Yaskawa INFORM job: SKRZYNIA_5340_-90_STOPNI_10BR.JBI

/JOB
//NAME SKRZYNIA_5340_-90_STOPNI_10BR
///FOLDERNAME 02-SKRZYNIE_JOBS
//POS
///NPOS 695,695,0,50,0,0
///TOOL 0
///POSTYPE PULSE
///PULSE
C00000=0,-52280,40443,0,6876,0
C00001=-82314,-24956,17040,-59626,-27382,-6248
C00002=-93910,-8625,17040,-59626,-43355,-6248
C00003=-98846,-1061,-42166,-80308,-57081,16120
C00004=-100452,6057,-48127,-85711,-56704,21322
C00005=-96957,25597,-37888,-85158,-62082,25522
C00006=-95580,33075,-33256,-84644,-64024,26851
C00007=-94380,33739,-32188,-85134,-63496,26721
C00008=-95580,33075,-33256,-84644,-64024,26851
C00009=-94940,31262,-36138,-85248,-63712,27160
C00010=-95580,33075,-33256,-84644,-64024,26851
C00011=-95263,33142,-33256,-84677,-63995,26850
C00012=-95263,33142,-33256,-84677,-63995,26850
C00013=-94261,33702,-32359,-85087,-63552,26740
C00014=-95263,33142,-33256,-84677,-63995,26850
C00015=-94777,31773,-35433,-85135,-63758,27084
C00016=-95263,33142,-33256,-84677,-63995,26850
C00017=-95260,33144,-33256,-84678,-63995,26850
C00018=-95260,33144,-33256,-84678,-63995,26850
C00019=-94282,33689,-32380,-85076,-63563,26742
C00020=-95260,33144,-33256,-84678,-63995,26850
C00021=-94827,31920,-35204,-85086,-63784,27059
C00022=-95260,33144,-33256,-84678,-63995,26850
C00023=-95258,33145,-33257,-84676,-63996,26846
C00024=-95258,33145,-33257,-84676,-63996,26846
C00025=-94286,33686,-32387,-85074,-63568,26738
C00026=-95258,33145,-33257,-84676,-63996,26846
C00027=-94874,32057,-34990,-85039,-63809,27032
C00028=-95258,33145,-33257,-84676,-63996,26846
C00029=-95258,33145,-33257,-84676,-63996,26846
C00030=-95258,33145,-33257,-84676,-63996,26846
C00031=-94323,33667,-32422,-85059,-63584,26741
C00032=-95258,33145,-33257,-84676,-63996,26846
C00033=-94899,32130,-34875,-85014,-63820,27019
C00034=-95258,33145,-33257,-84676,-63996,26846
C00035=-95258,25631,32269,-66559,-75499,2416
C00036=-95258,25631,32269,-66559,-75499,2416
C00037=-94333,26371,33350,-66433,-74983,2224
C00038=-95258,25631,32269,-66559,-75499,2416
C00039=-94886,24142,30119,-66602,-75133,2534
C00040=-95258,25631,32269,-66559,-75499,2416
C00041=-98646,19496,-17631,-99827,-80462,21224
C00042=-98811,21047,-15512,-99242,-81394,20987
C00043=-97886,21574,-14788,-99528,-80824,20997
C00044=-98811,21047,-15512,-99242,-81394,20987
C00045=-98517,19954,-17009,-99363,-81263,21101
C00046=-98811,21047,-15512,-99242,-81394,20987
C00047=-98811,19937,1242,-97498,-78933,15296
C00048=-98811,19937,1242,-97498,-78933,15296
C00049=-97933,20465,1962,-97646,-78345,15298
C00050=-98811,19937,1242,-97498,-78933,15296
C00051=-98523,18806,-285,-97586,-78782,15407
C00052=-98811,19937,1242,-97498,-78933,15296
C00053=-99152,37522,67957,-90787,-75030,-95
C00054=-99152,37522,67957,-90787,-75030,-95
C00055=-98279,38495,69612,-90504,-74443,-274
C00056=-99152,37522,67957,-90787,-75030,-95
C00057=-98708,34478,62881,-90983,-74820,488
C00058=-99152,37522,67957,-90787,-75030,-95
C00059=-98988,22776,44546,-90608,-68570,2568
C00060=-94428,854,16076,-89248,-50738,4740
C00061=-88080,-20128,-3199,-80943,-31244,2335
C00062=-50003,-39410,-5978,-16260,-18649,-25999
C00063=-48287,-44591,-17414,-16172,-14532,-25809
C00064=-85348,-13130,13838,-41209,-47455,-8220
C00065=-99199,18818,35660,-68259,-73735,6208
C00066=-95720,11094,-10147,-77005,-64537,18127
C00067=-95720,11099,-9975,-76955,-64559,18070
C00068=-97322,30100,38585,-71742,-79662,10416
C00069=-96349,30901,39804,-71630,-79090,10224
C00070=-97322,30100,38585,-71742,-79662,10416
C00071=-97054,28837,36680,-71776,-79387,10556
C00072=-97322,30100,38585,-71742,-79662,10416
C00073=-97373,30352,38967,-71736,-79717,10385
C00074=-97373,30352,38967,-71736,-79717,10385
C00075=-96432,31128,40151,-71627,-79165,10198
C00076=-97373,30352,38967,-71736,-79717,10385
C00077=-97071,28917,36802,-71776,-79407,10544
C00078=-97373,30352,38967,-71736,-79717,10385
C00079=-97356,30262,38827,-71739,-79698,10398
C00080=-97356,30262,38827,-71739,-79698,10398
C00081=-96507,30957,39891,-71642,-79201,10230
C00082=-97356,30262,38827,-71739,-79698,10398
C00083=-97092,29010,36937,-71773,-79425,10538
C00084=-97356,30262,38827,-71739,-79698,10398
C00085=-97431,30641,39402,-71725,-79780,10352
C00086=-97431,30641,39402,-71725,-79780,10352
C00087=-96578,31348,40481,-71627,-79280,10181
C00088=-97431,30641,39402,-71725,-79780,10352
C00089=-97114,29116,37095,-71767,-79448,10523
C00090=-97431,30641,39402,-71725,-79780,10352
C00091=-99739,25677,21114,-82085,-78790,-4409
C00092=-99739,25677,21114,-82085,-78790,-4409
C00093=-98872,26250,21941,-82102,-78216,-4501
C00094=-99739,25677,21114,-82085,-78790,-4409
C00095=-99422,24232,19045,-82158,-78544,-4261
C00096=-99739,25677,21114,-82085,-78790,-4409
C00097=-98070,21699,18791,-100677,-76082,-5031
C00098=-98401,27942,27737,-100067,-79473,-6121
C00099=-97586,28537,28617,-100081,-78897,-6135
C00100=-98401,27942,27737,-100067,-79473,-6121
C00101=-98064,26400,25481,-100144,-79339,-5917
C00102=-98401,27942,27737,-100067,-79473,-6121
C00103=-99160,29228,35009,-99418,-79080,-8034
C00104=-98369,30564,38686,-99156,-78226,-8682
C00105=-97572,31199,39655,-99108,-77655,-8715
C00106=-98369,30564,38686,-99156,-78226,-8682
C00107=-98044,28949,36247,-99232,-78106,-8445
C00108=-98369,30564,38686,-99156,-78226,-8682
C00109=-99160,29228,35009,-99418,-79080,-8034
C00110=-98369,30564,38686,-99156,-78226,-8682
C00111=-97572,31199,39655,-99108,-77655,-8715
C00112=-98369,30564,38686,-99156,-78226,-8682
C00113=-98044,28949,36247,-99232,-78106,-8445
C00114=-98369,30564,38686,-99156,-78226,-8682
C00115=-91461,-11352,-34112,-115843,-54659,7933
C00116=-98486,-14751,-40891,-114294,-59712,7739
C00117=-84089,-24462,-58822,-138905,-52068,17717
C00118=-93370,-29108,-64994,-133695,-56362,15444
C00119=-62749,-65297,-81682,-146767,-31843,20298
C00120=-73187,-23116,26488,-26118,-57509,-28469
C00121=-99665,-12992,-24886,-73613,-54905,-950
C00122=-98398,-8109,-25057,-81551,-55130,4513
C00123=-99451,17861,2757,-80571,-73406,6045
C00124=-99819,33446,48735,-87787,-79679,-1235
C00125=-99819,33446,48735,-87787,-79679,-1235
C00126=-98945,34179,49898,-87659,-79086,-1350
C00127=-99819,33446,48735,-87787,-79679,-1235
C00128=-99591,32133,46677,-87830,-79529,-1033
C00129=-99819,33446,48735,-87787,-79679,-1235
C00130=-98853,28116,28355,-96898,-79749,4777
C00131=-98853,30464,37910,-96149,-78952,2546
C00132=-98284,30904,38579,-96116,-78548,2515
C00133=-98853,30464,37910,-96149,-78952,2546
C00134=-98656,29478,36421,-96191,-78865,2688
C00135=-98853,30464,37910,-96149,-78952,2546
C00136=-94437,3365,15121,-90804,-55123,21
C00137=-76606,-19838,2636,-59027,-23020,-13375
C00138=-49667,-45532,-21960,-5654,-17518,-35856
C00139=-47485,-50287,-32535,-1070,-13732,-37871
C00140=-36103,-65917,11738,-26975,4295,7905
C00141=6327,-52297,40484,-8600,6957,5944
C00142=0,-52280,40443,0,6876,0
C00143=0,-52280,40443,0,6876,0
C00144=0,-43112,23163,32261,-40956,29092
C00145=-48283,-21883,28214,-25170,-26491,48363
C00146=-46664,-3144,58041,-18842,-32105,45325
C00147=-50347,-18571,12268,-49104,-16423,60029
C00148=-53571,-17125,12073,-56866,-17385,63433
C00149=-52069,-15730,13206,-55612,-16432,62999
C00150=-53474,-15384,13495,-57637,-17161,63825
C00151=-53571,-17125,12073,-56866,-17385,63433
C00152=-50509,-19000,10610,-51503,-15997,61182
C00153=-53130,-17211,12007,-56251,-17152,63186
C00154=-51822,-15992,12994,-55136,-16324,62798
C00155=-53635,-15431,13457,-57815,-17251,63894
C00156=-53130,-17211,12007,-56251,-17152,63186
C00157=-50704,-18403,11069,-52157,-16018,61478
C00158=-53231,-16470,14622,-53206,-17893,61673
C00159=-51756,-15101,15744,-51790,-16990,61165
C00160=-53741,-14453,16285,-54808,-17949,62397
C00161=-53231,-17580,11714,-56182,-17246,63139
C00162=-51814,-19410,10295,-53186,-16720,61844
C00163=-53629,-18979,7405,-62018,-16535,65958
C00164=-52238,-17698,8415,-61175,-15613,65699
C00165=-53551,-17401,8655,-62910,-16346,66402
C00166=-52880,-17654,11656,-55678,-17066,62935
C00167=-51005,-17995,11387,-52847,-16122,61778
C00168=-52964,-17611,11689,-55811,-17106,62990
C00169=-51611,-16353,12697,-54642,-16249,62582
C00170=-53495,-15765,13180,-57466,-17201,63739
C00171=-52964,-17611,11689,-55811,-17106,62990
C00172=-51030,-17982,11395,-52891,-16135,61798
C00173=-52975,-17563,11726,-55850,-17109,63009
C00174=-51607,-16289,12749,-54669,-16241,62596
C00175=-53283,-15811,13140,-57177,-17094,63622
C00176=-52975,-17563,11726,-55850,-17109,63009
C00177=-50945,-18019,11363,-52741,-16103,61737
C00178=-52728,-17788,11545,-55393,-17010,62816
C00179=-51045,-16207,12813,-53894,-15944,62287
C00180=-52895,-15647,13274,-56746,-16874,63461
C00181=-52728,-17788,11545,-55393,-17010,62816
C00182=-50945,-18019,11363,-52741,-16103,61737
C00183=-52556,-17520,11756,-55311,-16888,62798
C00184=-51113,-16157,12849,-54025,-15975,62343
C00185=-52730,-15718,13210,-56498,-16792,63358
C00186=-52556,-17520,11756,-55311,-16888,62798
C00187=-50945,-18019,11363,-52741,-16103,61737
C00188=-51893,-17787,11546,-54246,-16568,62356
C00189=-50379,-16341,12703,-52826,-15610,61849
C00190=-52406,-15704,13225,-56071,-16614,63190
C00191=-51893,-17787,11546,-54246,-16568,62356
C00192=-50028,-22953,-3957,-22347,-31919,54220
C00193=-50947,-22502,-3625,-23433,-32061,54736
C00194=-49421,-20951,-2455,-21951,-31329,54057
C00195=-51207,-20433,-2055,-24026,-31698,55041
C00196=-50529,-22709,-3778,-22940,-31995,54502
C00197=-49763,-25421,-36239,-24565,-26935,60445
C00198=-49763,-25421,-36239,-24565,-26935,60445
C00199=-48299,-23485,-34758,-23276,-26122,59713
C00200=-50218,-22723,-34165,-25568,-26529,60993
C00201=-49763,-25421,-36239,-24565,-26935,60445
C00202=-50713,-12366,-58367,-41124,-17813,74400
C00203=-50824,-12254,-58263,-41255,-17847,74484
C00204=-49431,-10052,-56192,-40383,-17131,73813
C00205=-50915,-9358,-55524,-41955,-17664,74847
C00206=-51028,-12852,-58814,-41301,-17980,74542
C00207=-49763,-25421,-36239,-24565,-26935,60445
C00208=-50529,-22709,-3778,-22940,-31995,54502
C00209=-45389,-28224,4312,-35967,-15579,54278
C00210=-40154,-51179,-915,-24203,-8234,36524
C00211=0,-52280,40443,0,6876,0
C00212=0,-52280,40443,0,6876,0
C00213=-2117,-50103,-33543,-4117,45077,85249
C00214=26439,-48928,-33543,-4117,-52362,85249
C00215=26439,-27355,-33543,-41485,-52362,85249
C00216=39218,-24492,-41653,-51934,-39374,86964
C00217=39218,-24492,-41653,-51934,-39374,86964
C00218=46639,7575,-9331,-26045,-41627,82486
C00219=47278,8641,-9483,-26175,-40625,82510
C00220=46369,10567,-7126,-26545,-41054,82831
C00221=47278,8641,-9483,-26175,-40625,82510
C00222=48256,9506,-8430,-25641,-40400,82076
C00223=47278,8641,-9483,-26175,-40625,82510
C00224=44522,-635,-31983,-49264,-28311,89687
C00225=44247,-628,-31975,-49394,-28443,89790
C00226=43310,1314,-29842,-49807,-28910,90140
C00227=44247,-628,-31975,-49394,-28443,89790
C00228=45313,152,-31124,-48894,-27920,89380
C00229=44247,-628,-31975,-49394,-28443,89790
C00230=41572,-13073,-22520,-50760,-38355,84033
C00231=21909,-6773,-14577,-94161,-56302,89381
C00232=23773,-3183,-10897,-94486,-55065,89563
C00233=24904,-823,-8382,-94654,-54308,89644
C00234=24395,1151,-6219,-94590,-54651,89617
C00235=24904,-823,-8382,-94654,-54308,89644
C00236=26178,-337,-7854,-94816,-53451,89710
C00237=24904,-823,-8382,-94654,-54308,89644
C00238=17020,-16061,-23281,-93084,-59494,88637
C00239=-21568,-26506,-31664,-90508,-85573,86639
C00240=-8557,-39769,-22319,-51419,-69406,84680
C00241=-8557,-39769,-22319,-51419,-69406,84680
C00242=32994,-9735,-10751,-29019,-59471,69498
C00243=43974,9628,-22604,-36190,-36396,73426
C00244=45932,13115,-22315,-37472,-33732,73846
C00245=45228,14664,-20329,-37571,-34159,74020
C00246=45932,13115,-22315,-37472,-33732,73846
C00247=46653,13731,-21526,-37109,-33514,73520
C00248=45932,13115,-22315,-37472,-33732,73846
C00249=39039,866,-6986,-42761,-44691,67687
C00250=30717,-9248,-22721,-77433,-42696,79486
C00251=32434,-7077,-20587,-77571,-41526,79457
C00252=31883,-5576,-19073,-77676,-41878,79560
C00253=32434,-7077,-20587,-77571,-41526,79457
C00254=33092,-6769,-20280,-77576,-41084,79417
C00255=32434,-7077,-20587,-77571,-41526,79457
C00256=30527,-14106,-27266,-76898,-42917,79150
C00257=25454,-9581,-17335,-94425,-53880,89429
C00258=24965,-2445,-10120,-94645,-54263,89631
C00259=24893,-1278,-8874,-94650,-54314,89639
C00260=24417,557,-6877,-94595,-54636,89618
C00261=24893,-1278,-8874,-94650,-54314,89639
C00262=25752,-956,-8526,-94759,-53737,89684
C00263=24893,-1278,-8874,-94650,-54314,89639
C00264=23817,-1527,-9142,-94518,-55040,89587
C00265=24871,-1152,-8735,-94651,-54328,89643
C00266=24440,508,-6926,-94601,-54619,89624
C00267=24871,-1152,-8735,-94651,-54328,89643
C00268=25635,-865,-8427,-94748,-53815,89684
C00269=24871,-1152,-8735,-94651,-54328,89643
C00270=33203,-4295,-13750,-123758,-49995,81034
C00271=35028,4195,-6818,-132965,-58836,87950
C00272=35028,4195,-6818,-132965,-58836,87950
C00273=34452,5837,-4911,-132720,-59045,87770
C00274=35028,4195,-6818,-132965,-58836,87950
C00275=35710,4593,-6360,-133217,-58512,88125
C00276=35028,4195,-6818,-132965,-58836,87950
C00277=24762,-11408,-28656,-113055,-60293,85383
C00278=-28645,-26349,-41223,-103369,-91870,78302
C00279=-28645,-26349,-41223,-103369,-91870,78302
C00280=-25549,-24286,-26215,-66769,-87032,80148
C00281=27561,-8271,-12315,-63268,-52553,74387
C00282=29336,-165,-3925,-63163,-51316,74265
C00283=29518,765,-2904,-63127,-51205,74233
C00284=28850,2962,-447,-63227,-51636,74327
C00285=29518,765,-2904,-63127,-51205,74233
C00286=30662,1292,-2320,-62902,-50501,74035
C00287=29518,765,-2904,-63127,-51205,74233
C00288=30773,10953,32136,-106912,-46141,83783
C00289=30773,10953,32136,-106912,-46141,83783
C00290=30080,13410,35293,-106601,-46463,83481
C00291=30773,10953,32136,-106912,-46141,83783
C00292=32007,11622,32987,-106899,-45346,83915
C00293=30773,10953,32136,-106912,-46141,83783
C00294=28321,-8642,-16372,-95739,-47180,89965
C00295=28583,-7344,-15096,-95864,-47019,90043
C00296=27897,-5229,-12965,-95873,-47499,90079
C00297=28583,-7344,-15096,-95864,-47019,90043
C00298=29900,-6813,-14567,-96101,-46141,90154
C00299=28583,-7344,-15096,-95864,-47019,90043
C00300=27852,-7537,-15286,-95742,-47508,89986
C00301=28448,-7306,-15058,-95845,-47110,90035
C00302=27795,-5283,-13021,-95851,-47567,90065
C00303=28448,-7306,-15058,-95845,-47110,90035
C00304=29772,-6774,-14527,-96083,-46226,90146
C00305=28448,-7306,-15058,-95845,-47110,90035
C00306=18552,-19531,-26179,-93438,-53589,88597
C00307=40301,-14999,-52277,-148979,-69262,86714
C00308=42323,-33,-37432,-150113,-69667,87489
C00309=53245,19091,3515,-165691,-72595,90030
C00310=53641,19552,4138,-165817,-72473,90151
C00311=53058,20743,5761,-165615,-72317,89948
C00312=53641,19552,4138,-165817,-72473,90151
C00313=54155,20160,4967,-165982,-72308,90306
C00314=53641,19552,4138,-165817,-72473,90151
C00315=23439,-10154,-17205,-109204,-58547,76547
C00316=2382,-21913,-40813,-107544,-74451,77239
C00317=-31257,-15877,-35733,-102288,-96107,74463
C00318=-39204,-18003,-7668,-86141,-99190,68413
C00319=-5592,-5690,18047,-75373,-79525,63129
C00320=19039,-439,25862,-68224,-64120,61443
C00321=21624,5223,26011,-69375,-61155,63193
C00322=24437,11840,34139,-68260,-59598,62567
C00323=24053,13588,36402,-68249,-59917,62491
C00324=24437,11840,34139,-68260,-59598,62567
C00325=25079,12112,34488,-68051,-59212,62472
C00326=24437,11840,34139,-68260,-59598,62567
C00327=21370,4935,25667,-69451,-61310,63230
C00328=-18351,-11002,3811,-80352,-86206,66275
C00329=-34619,-5846,8788,-82342,-97004,67025
C00330=-40684,-19963,-8478,-86482,-100204,67987
C00331=1570,-13136,-5998,-86227,-71173,69099
C00332=13966,-6596,-2340,-86587,-62612,70052
C00333=24093,-1862,-9504,-94546,-54850,89594
C00334=24093,-1862,-9504,-94546,-54850,89594
C00335=23519,425,-7024,-94488,-55240,89573
C00336=24093,-1862,-9504,-94546,-54850,89594
C00337=25256,-1442,-9053,-94693,-54067,89656
C00338=24093,-1862,-9504,-94546,-54850,89594
C00339=27718,4364,12871,-105518,-51077,86669
C00340=27718,4364,12871,-105518,-51077,86669
C00341=27164,6353,15202,-105385,-51398,86539
C00342=27718,4364,12871,-105518,-51077,86669
C00343=28828,4851,13441,-105618,-50355,86801
C00344=27718,4364,12871,-105518,-51077,86669
C00345=20930,-1364,27707,-95004,-52134,77785
C00346=-41463,-32191,18163,-91991,-64949,55938
C00347=0,-52277,40442,0,6872,4
C00348=-82314,-24956,17040,-59626,-27382,-6248
C00349=-93910,-8625,17040,-59626,-43355,-6248
C00350=-98846,-1061,-42166,-80308,-57081,16120
C00351=-100452,6057,-48127,-85711,-56704,21322
C00352=-95564,34698,-34234,-85516,-63941,27819
C00353=-94221,34299,-28769,-82558,-65564,25844
C00354=-94107,37241,-30442,-84005,-65307,27544
C00355=-95103,32620,-31323,-83378,-64939,26072
C00356=-95103,32620,-31323,-83378,-64939,26072
C00357=-93990,32828,-31380,-83932,-64473,26160
C00358=-94063,31710,-30585,-83283,-64598,25457
C00359=-96692,32939,-31211,-82617,-65723,26190
C00360=-96111,21840,170,-71736,-70232,11396
C00361=-94229,22391,773,-71789,-70557,11468
C00362=-94283,22521,1025,-71678,-70686,11433
C00363=-95675,19167,-4176,-72970,-68231,11735
C00364=-95681,24338,3488,-71459,-71669,11415
C00365=-94245,22750,1246,-71757,-70674,11453
C00366=-94341,22923,1499,-71729,-70746,11440
C00367=-96213,24222,3324,-71394,-71999,11479
C00368=-95517,23330,2066,-71543,-71508,11507
C00369=-94304,22892,1449,-71738,-70721,11443
C00370=-94158,22889,1452,-71756,-70627,11429
C00371=-96071,24319,3461,-71408,-71916,11455
C00372=-96941,-6406,-33809,-76117,-54125,10511
C00373=-89093,-33107,-44597,-67545,-52550,2722
C00374=-66103,-61757,7450,-21008,-32955,-5749
C00375=4223,-52290,40457,-5766,6913,3980
C00376=4223,-52290,40457,-5766,6913,3980
C00377=-4538,-50065,-33535,-3011,44998,84219
C00378=24207,-49248,-33668,-5551,-52644,86091
C00379=25094,-27722,-33812,-41887,-53054,85599
C00380=38036,-25052,-42086,-52219,-40087,87228
C00381=37328,-2824,-24733,-57182,-37821,90318
C00382=36700,-2520,-13735,-51589,-42201,86442
C00383=37520,2330,-3498,-48550,-43875,84431
C00384=37520,1020,-12079,-52650,-40851,87066
C00385=48458,-261,-12985,-24069,-43340,80504
C00386=36153,7296,-1758,-40139,-50302,89334
C00387=37146,11264,2520,-40849,-50296,89553
C00388=38059,11410,-1863,-40565,-47910,90206
C00389=36726,6476,-7858,-41213,-48206,90783
C00390=19339,7883,9818,-77509,-64249,74140
C00391=19027,1888,-16187,-103553,-67480,82955
C00392=24158,3537,-14322,-106039,-60939,84018
C00393=24143,4321,-7309,-103852,-59670,81875
C00394=19531,2904,-8928,-102027,-65985,80961
C00395=20232,-3383,-14682,-86495,-63009,78978
C00396=-24375,-51634,-49601,-83793,-94064,73950
C00397=4223,-52290,40457,-5766,6913,3980
C00398=-4825,-36686,24602,37792,-30278,35378
C00399=-46221,-29633,7403,-27051,-24124,46751
C00400=-46221,-29633,7403,-27051,-24124,46751
C00401=-52474,-20611,11454,-41004,-23045,52959
C00402=-60257,-19980,-2088,-84190,-23320,82051
C00403=-63868,-19883,-6318,-95759,-28031,88346
C00404=-51819,-22965,8574,-41365,-22900,53139
C00405=-4825,-36686,24602,37792,-30278,35378
C00406=0,-52280,40443,0,6876,0
C00407=4223,-52290,40457,-5766,6913,3980
C00408=-66103,-61757,7450,-21008,-32955,-5749
C00409=-89093,-33107,-44597,-67545,-52550,2722
C00410=-96941,-6406,-33809,-76117,-54125,10511
C00411=-99429,14378,84,-80785,-71596,8628
C00412=-99699,24313,24829,-82602,-77917,4569
C00413=-98066,26841,20697,-83331,-79245,6860
C00414=-98079,26929,20513,-83349,-79351,6953
C00415=-99638,19663,10292,-84193,-74452,7551
C00416=-99636,19665,10291,-84197,-74448,7550
C00417=-98131,26698,20177,-83371,-79212,6975
C00418=-98097,25980,12653,-84102,-79057,9159
C00419=-99636,19665,10291,-84197,-74448,7550
C00420=-99636,19665,10291,-84197,-74448,7550
C00421=-98186,26934,20517,-83350,-79332,6954
C00422=-98240,27087,20738,-83333,-79465,6940
C00423=-99636,19665,10291,-84197,-74448,7550
C00424=-99215,3992,8526,-80547,-63068,1835
C00425=-100264,1107,23397,-72827,-59854,-5092
C00426=-100264,1107,23397,-72827,-59854,-5092
C00427=-99514,-9483,18258,-71284,-60958,-4118
C00428=-61441,-38616,11032,-55510,-42874,-3049
C00429=4223,-52290,40457,-5766,6913,3980
C00430=-22331,-23394,-30093,-82917,-82006,85712
C00431=22434,-14401,-3235,-51104,-60845,74728
C00432=42744,21307,45077,-24753,-69813,65333
C00433=33655,14083,18147,-45417,-58301,71861
C00434=33641,11943,8279,-47835,-54840,73983
C00435=36574,13250,23432,-35354,-61822,69159
C00436=28497,326,20939,-70981,-47632,72427
C00437=30972,5983,29862,-68494,-46670,70994
C00438=31029,11571,45127,-63398,-49004,67378
C00439=28971,8096,39948,-65070,-49810,68216
C00440=29759,-12862,-24221,-91747,-41905,86600
C00441=35278,-10419,-21940,-93284,-36771,87139
C00442=36208,-10883,-22374,-93618,-35345,87231
C00443=27219,-23595,-33313,-89555,-43517,85303
C00444=10564,-40773,-45889,-85382,-54876,82708
C00445=-14984,-61618,-24572,-87392,-53367,60735
C00446=9346,-67436,-18786,-75708,-34590,53709
C00447=40938,-55232,35946,-9746,5421,6718
C00448=4223,-52290,40457,-5766,6913,3980
C00449=-4825,-36686,24602,37792,-30278,35378
C00450=-46221,-29633,7403,-27051,-24124,46751
C00451=-56796,-22932,368,-68953,-21567,70907
C00452=-61611,-20349,-6598,-95791,-25091,88405
C00453=-63740,-19715,-7390,-98604,-28245,90373
C00454=-52085,-22687,8760,-40927,-22666,52970
C00455=-49294,-34086,9663,-30689,-30758,52546
C00456=4223,-52290,40457,-5766,6913,3980
C00457=0,-52280,40443,0,6876,0
C00458=0,-52280,40443,0,6876,0
C00459=-61754,-61602,7279,-16215,-32140,-7126
C00460=-89313,-24027,20291,-53466,-58905,-4975
C00461=-97807,-25409,-21837,-78881,-62828,2121
C00462=-95644,-21015,-18476,-76474,-46020,1039
C00463=-99784,20282,11129,-84157,-74554,7499
C00464=-100058,25789,39872,-88643,-74345,1113
C00465=-98402,30585,40634,-89771,-78826,2411
C00466=-98157,28480,31016,-94616,-79375,5454
C00467=-99711,20530,18234,-96341,-74733,7105
C00468=-100058,25789,39872,-88643,-74345,1113
C00469=-98402,30585,40634,-89771,-78826,2411
C00470=-98157,28480,31016,-94616,-79375,5454
C00471=-99711,20530,18234,-96341,-74733,7105
C00472=-99082,-18510,-57081,-109378,-57172,19856
C00473=-62624,-58412,-72925,-116868,-19429,18539
C00474=-75165,-16680,32803,-38944,-52307,-27215
C00475=-75165,-16680,32803,-38944,-52307,-27215
C00476=-96391,11374,61850,-52875,-60261,-22353
C00477=-96391,-17993,-25254,-79577,-45337,-1997
C00478=-84714,-13514,-21320,-79690,-37366,-2300
C00479=-92093,-5454,-13554,-80916,-52292,-613
C00480=-99761,24721,23429,-79408,-77929,-316
C00481=-100093,22783,4772,-83722,-77198,5432
C00482=-98451,25119,10323,-84368,-78687,2343
C00483=-98528,26732,19657,-84000,-79459,-654
C00484=-100109,23919,19160,-82044,-77303,1139
C00485=-98037,-4340,-16930,-86109,-58746,2389
C00486=-93345,-31758,-40240,-83703,-37467,-946
C00487=-81087,-35886,-14825,-53529,-36311,-18004
C00488=-47029,-49867,-20464,-11808,-29290,-36568
///LIMIT ON
C00489=-41431,-67449,10869,-1325,127,-6150
///LIMIT OFF
C00490=6328,-52297,40483,-8599,6957,5944
C00491=-8648,-69005,-18270,-84275,-43232,53472
C00492=18757,-59462,-34892,-84638,-37529,67311
C00493=26772,-23733,-33422,-89486,-43820,85275
C00494=29039,-10071,-21608,-91386,-45181,86629
C00495=29639,-5923,-17523,-91591,-45648,86808
C00496=29709,-5453,-17046,-91618,-45636,86826
C00497=29138,-10182,-21714,-91372,-45196,86624
C00498=20424,-22725,-32635,-88800,-51006,85261
C00499=28416,-11420,-25238,-98178,-46636,84572
C00500=30481,-6584,-16425,-92636,-44382,82541
C00501=30464,-7521,-23523,-96665,-44944,85234
C00502=28416,-11420,-25238,-98178,-46636,84572
C00503=-23524,-33387,-42654,-89891,-81168,80229
C00504=-23524,-33387,-42654,-89891,-81168,80229
C00505=33935,-6399,-10013,-60506,-43064,77980
C00506=34878,-3211,-6740,-60356,-42422,77865
C00507=34873,-3218,-6748,-60357,-42424,77868
C00508=33935,-6399,-10013,-60506,-43064,77980
C00509=17782,-19597,1250,-60925,-51448,69151
C00510=-243,-43047,-13224,-69794,-55957,65877
C00511=42700,-55269,36176,-13619,5333,9062
C00512=6328,-52297,40483,-8599,6957,5944
C00513=-10231,-60460,6271,71658,-11927,-13637
C00514=-49129,-39322,3023,-34904,-18609,43900
C00515=-57258,-19535,13114,-46502,-25798,55150
C00516=-58736,-19151,1344,-78268,-22199,76919
C00517=-56868,-17231,8572,-62431,-21728,66645
C00518=-56011,-29317,6725,-41009,-27363,52457
C00519=-10137,-60963,4526,62308,-14518,-6745
C00520=0,-52280,40443,0,6876,0
C00521=0,-52280,40443,0,6876,0
C00522=-41653,-63035,2931,-3578,-7576,-14589
C00523=-45770,-50109,-20524,-10089,-29273,-37310
C00524=-80544,-36303,-15042,-52975,-36116,-18265
C00525=-93028,-32302,-40599,-83495,-37263,-1079
C00526=-98446,-3141,-15678,-86094,-59021,2414
C00527=-99951,24070,19376,-82000,-77829,1145
C00528=-98655,27908,24922,-81730,-79774,792
C00529=-98593,28720,26118,-81685,-80145,709
C00530=-99951,24070,19376,-82000,-77829,1145
C00531=-99951,24070,19376,-82000,-77829,1145
C00532=-98577,27118,23759,-81796,-79157,859
C00533=-98518,28577,26461,-81649,-79882,537
C00534=-99951,24070,19376,-82000,-77829,1145
C00535=-99951,24070,19376,-82000,-77829,1145
C00536=-98479,26563,22955,-81844,-78651,906
C00537=-98651,28095,26058,-81646,-79654,489
C00538=-99951,24070,19376,-82000,-77829,1145
C00539=-97595,-1409,-12320,-84284,-60474,1798
C00540=-100010,-16422,-27011,-84227,-53565,945
C00541=-88098,-29848,-22776,-71580,-48483,-7812
C00542=-81694,-37220,-20464,-64791,-45723,-12569
C00543=-45770,-50109,-20524,-10089,-29273,-37310
C00544=-40984,-65135,6743,-2520,-4051,-10897
C00545=0,-52280,40443,0,6876,0
C00546=40939,-55232,35946,-9746,5421,6719
C00547=8707,-69002,-18268,-75213,-34271,52581
C00548=23267,-58917,-25142,-81990,-31707,62852
C00549=27307,-5613,10331,-81857,-46454,76095
C00550=30064,-5598,-963,-91827,-44222,81590
C00551=30419,-1725,5291,-88668,-43977,80354
C00552=30554,-300,10432,-88528,-43656,79164
C00553=29815,-6351,-3652,-90193,-44535,81892
C00554=29567,1847,27834,-65726,-48411,69959
C00555=23257,11670,30420,-81328,-57342,77033
C00556=23257,16856,45442,-77525,-58254,73578
C00557=21577,7912,33836,-78698,-59121,74340
C00558=17856,-9033,24892,-70658,-55966,67475
C00559=20838,-7097,2019,-111788,-62648,79114
C00560=40635,280,-7982,-142398,-56681,90238
C00561=32653,-9455,434,-90251,-40347,77213
C00562=40635,572,-6271,-142064,-55879,89947
C00563=40665,7761,2001,-141975,-55632,89869
C00564=40707,9678,10648,-140211,-51894,88431
C00565=39416,1907,3178,-139370,-51839,87774
C00566=7767,-21333,-19174,-120411,-69473,77116
C00567=33666,-18553,20064,-54519,-41956,59729
C00568=4032,-43511,13506,-33366,-30942,40837
C00569=22997,-56875,21315,16958,-8102,3163
C00570=0,-52280,40443,0,6876,0
C00571=-50974,-46557,23391,-77768,-13896,42026
C00572=-53474,-39983,4253,-39182,-18848,44272
C00573=-56619,-19856,12878,-45665,-25558,54806
C00574=-53298,-26712,-11188,-26889,-32979,52528
C00575=-57200,-20845,-7559,-37425,-33513,53351
C00576=-58648,-23818,-25853,-45100,-31207,62168
C00577=-58477,-22145,-38977,-48305,-29254,64725
C00578=-51868,-27423,-11673,-25269,-32728,51737
C00579=-49121,-45409,-2608,-26656,-19965,38583
C00580=-21301,-61008,4568,43957,-10534,-712
C00581=0,-52280,40443,0,6876,0
C00582=0,-52280,40443,0,6876,0
C00583=-40221,-67507,11044,-1325,-65,-6716
C00584=-45770,-50109,-20525,-10088,-29274,-37311
C00585=-80544,-36303,-15042,-52975,-36116,-18265
C00586=-93028,-32301,-40599,-83495,-37262,-1079
C00587=-97841,-4898,-17503,-86112,-58614,2374
C00588=-98519,17635,7561,-106659,-77043,7343
C00589=-96245,23653,15791,-106069,-78604,6508
C00590=-96042,26225,19489,-105739,-79656,6032
C00591=-98519,17635,7561,-106659,-77043,7343
C00592=-98519,17635,7561,-106659,-77043,7343
C00593=-96298,25666,18652,-105800,-79560,6117
C00594=-95268,26547,15396,-109206,-81354,7908
C00595=-98519,17635,7561,-106659,-77043,7343
C00596=-96138,5697,-7380,-109479,-68538,9618
C00597=-100287,-3253,-24038,-111364,-68562,12025
C00598=-99412,-19117,-26908,-100833,-57247,5735
C00599=-91712,-30589,-22890,-72058,-50969,-7685
C00600=-81694,-37221,-20464,-64791,-45723,-12569
C00601=-45770,-50109,-20525,-10088,-29274,-37311
C00602=-40221,-67507,11044,-1325,-65,-6716
C00603=0,-52280,40443,0,6876,0
C00604=51241,-30653,28678,4016,-29070,6398
C00605=46185,-61941,-37286,-12736,-10732,51851
C00606=-13205,-44768,-23966,-65315,-59418,73750
C00607=-11120,-40541,-20876,-69249,-61539,75403
C00608=-836,-13033,12361,-83908,-73576,73378
C00609=18912,6214,32354,-79489,-60743,73080
C00610=21217,10898,38129,-78632,-59343,72736
C00611=23447,16313,45262,-77527,-58074,72177
C00612=23610,23756,64158,-73325,-59549,68283
C00613=18912,6214,32354,-79489,-60743,73080
C00614=-836,-13033,12361,-83908,-73576,73378
C00615=-20209,-39682,-20467,-71924,-67122,76479
C00616=-20209,-39682,-20467,-71924,-67122,76479
C00617=26353,-3691,11741,-61723,-54035,71160
C00618=29598,-2090,11073,-69087,-47235,76987
C00619=30217,-1844,4641,-75777,-45517,79979
C00620=29529,1742,11379,-68166,-49318,73572
C00621=24010,-9039,-4437,-79986,-50972,77255
C00622=24652,-10740,-12845,-99298,-50700,81949
C00623=28976,-2672,-4778,-100308,-47937,82653
C00624=31030,-2921,-9996,-112394,-49006,86348
C00625=24652,-10740,-12845,-99298,-50700,81949
C00626=-25637,-26222,-38592,-96633,-85474,81576
C00627=-36771,-16470,-4689,-95304,-89579,74076
C00628=-33704,-12343,7746,-85568,-87064,70052
C00629=4032,-43511,13506,-33366,-30942,40837
C00630=27500,-60047,23168,28912,-2679,-5784
C00631=0,-52280,40443,0,6876,0
C00632=-50971,-46557,23390,-77766,-13895,42026
C00633=-53475,-39984,4253,-39182,-18848,44273
C00634=-56619,-19856,12878,-45665,-25558,54806
C00635=-57643,-27958,-8553,-51854,-24771,59787
C00636=-66195,-24410,-19095,-90567,-31132,85904
C00637=-63290,-24193,-14362,-80030,-27547,78073
C00638=-39040,-40975,-15408,-18643,-21575,44866
C00639=-11647,-69843,-10959,56399,-11165,-4616
C00640=-15394,-57237,30542,-10392,5525,8219
C00641=0,-52280,40443,0,6876,0
C00642=0,-52280,40443,0,6876,0
///LIMIT ON
C00643=-40221,-67507,11044,-1325,-65,-6716
///LIMIT OFF
C00644=-45770,-50109,-20525,-10088,-29274,-37311
C00645=-95022,-19559,-3970,-66108,-42168,-11789
C00646=-84972,-7110,7117,-67721,-41324,-10731
C00647=-83869,-8155,6098,-67213,-40658,-10968
C00648=-99927,21772,-3530,-88309,-78218,7709
C00649=-97220,21950,1672,-79686,-74035,6807
C00650=-96918,21734,-3846,-80685,-73375,8528
C00651=-99839,23064,19027,-85806,-76881,822
C00652=-99839,23064,19027,-85806,-76881,822
C00653=-98572,26113,23382,-85571,-78492,509
C00654=-98656,28006,28806,-88976,-79248,97
C00655=-99839,24479,25828,-85077,-77001,-891
C00656=-99133,24879,24637,-94741,-77121,-2989
C00657=-98191,27052,27787,-94567,-78528,-3332
C00658=-98227,29022,36334,-93788,-77894,-5388
C00659=-100426,22466,21877,-95586,-77332,-2808
C00660=-99839,23064,19027,-85806,-76881,822
C00661=-86774,-13232,-16630,-85484,-41019,-1154
C00662=-97999,-21060,-29835,-88214,-48653,956
C00663=-98846,-3268,25064,-74217,-51189,-12584
C00664=-70313,-35289,-4922,-51188,-38634,-20596
C00665=-81694,-37221,-20464,-64791,-45723,-12569
C00666=-45770,-50109,-20525,-10088,-29274,-37311
C00667=-41628,-63095,3038,-3547,-7472,-14475
C00668=4223,-52290,40457,-5766,6913,3980
C00669=4224,-52288,40457,-5773,6909,3978
C00670=4224,-52288,40457,-28770,-64753,45638
C00671=6548,2882,44080,-77825,-67624,70557
C00672=22702,21750,69443,-66118,-61597,67582
C00673=25585,21999,63350,-62249,-61285,68688
C00674=25777,17209,50811,-62979,-59886,70957
C00675=23226,22825,71113,-65575,-61542,67353
C00676=24931,14697,51677,-80718,-51653,72069
C00677=24746,14409,39758,-87518,-53542,76879
C00678=24784,21556,58944,-82031,-53873,72431
C00679=22657,12722,42993,-85587,-54940,74916
C00680=-4427,-20395,-7318,-104668,-69521,79317
C00681=768,-20151,-3587,-97758,-65802,76626
C00682=-14736,-21545,-1233,-93598,-60476,72578
C00683=1642,-46684,14475,-47609,-24983,34912
C00684=27500,-60047,23168,28912,-2679,-5784
C00685=0,-52280,40443,0,6876,0
C00686=-50971,-46557,23390,-77766,-13895,42026
C00687=-53475,-39984,4253,-39182,-18848,44273
C00688=-56619,-19856,12878,-45665,-25558,54806
C00689=-53891,-17708,14512,-43170,-23995,53902
C00690=-60674,-17500,6427,-71116,-24772,71097
C00691=-63181,-17997,2063,-82122,-26831,78394
C00692=-39402,-27697,7664,-17904,-21663,43170
C00693=-11647,-69843,-10959,56399,-11165,-4616
C00694=0,-52280,40443,0,6876,0
BC00000=464364
BC00001=445130
BC00002=445130
BC00003=445130
BC00004=445130
BC00005=445130
BC00006=445130
BC00007=445130
BC00008=445130
BC00009=445130
BC00010=445130
BC00011=491232
BC00012=491232
BC00013=491232
BC00014=491232
BC00015=491232
BC00016=491232
BC00017=537442
BC00018=537442
BC00019=537442
BC00020=537442
BC00021=537442
BC00022=537442
BC00023=583546
BC00024=583546
BC00025=583546
BC00026=583546
BC00027=583546
BC00028=583546
BC00029=606594
BC00030=606594
BC00031=606594
BC00032=606594
BC00033=606594
BC00034=606594
BC00035=559393
BC00036=559393
BC00037=559393
BC00038=559393
BC00039=559393
BC00040=559393
BC00041=605503
BC00042=605503
BC00043=605504
BC00044=605503
BC00045=605503
BC00046=605503
BC00047=605503
BC00048=605503
BC00049=605503
BC00050=605503
BC00051=605503
BC00052=605503
BC00053=604255
BC00054=604255
BC00055=604255
BC00056=604255
BC00057=604255
BC00058=604255
BC00059=604255
BC00060=604255
BC00061=604255
BC00062=604255
BC00063=699121
BC00064=714117
BC00065=714117
BC00066=743139
BC00067=742930
BC00068=721797
BC00069=721797
BC00070=721797
BC00071=721797
BC00072=721797
BC00073=737203
BC00074=737203
BC00075=737203
BC00076=737203
BC00077=737203
BC00078=737203
BC00079=783275
BC00080=783275
BC00081=783275
BC00082=783275
BC00083=783275
BC00084=783275
BC00085=806364
BC00086=806364
BC00087=806364
BC00088=806364
BC00089=806364
BC00090=806364
BC00091=843190
BC00092=843190
BC00093=843190
BC00094=843190
BC00095=843190
BC00096=843190
BC00097=849204
BC00098=849204
BC00099=849204
BC00100=849204
BC00101=849204
BC00102=849204
BC00103=863801
BC00104=863801
BC00105=863801
BC00106=863801
BC00107=863801
BC00108=863801
BC00109=894523
BC00110=894523
BC00111=894523
BC00112=894523
BC00113=894523
BC00114=894523
BC00115=872244
BC00116=872244
BC00117=872244
BC00118=872244
BC00119=872244
BC00120=936612
BC00121=1007312
BC00122=1007425
BC00123=1007450
BC00124=973058
BC00125=973058
BC00126=973058
BC00127=973058
BC00128=973058
BC00129=973058
BC00130=988475
BC00131=988475
BC00132=988475
BC00133=988475
BC00134=988475
BC00135=988475
BC00136=976824
BC00137=970766
BC00138=986977
BC00139=935999
BC00140=857759
BC00141=811793
BC00142=811793
BC00143=811793
BC00144=811795
BC00145=919701
BC00146=919701
BC00147=949003
BC00148=951100
BC00149=951100
BC00150=951100
BC00151=951100
BC00152=889624
BC00153=889624
BC00154=889624
BC00155=889624
BC00156=889624
BC00157=828182
BC00158=828182
BC00159=828182
BC00160=828182
BC00161=828182
BC00162=766752
BC00163=766752
BC00164=766752
BC00165=766752
BC00166=766752
BC00167=705350
BC00168=705350
BC00169=705350
BC00170=705350
BC00171=705350
BC00172=643865
BC00173=643865
BC00174=643865
BC00175=643865
BC00176=643865
BC00177=582464
BC00178=582464
BC00179=582464
BC00180=582464
BC00181=582464
BC00182=520992
BC00183=520992
BC00184=520992
BC00185=520992
BC00186=520992
BC00187=459540
BC00188=459540
BC00189=459540
BC00190=459540
BC00191=459540
BC00192=459544
BC00193=459544
BC00194=459544
BC00195=459544
BC00196=459544
BC00197=459544
BC00198=459544
BC00199=459544
BC00200=459544
BC00201=459544
BC00202=459544
BC00203=459544
BC00204=459544
BC00205=459544
BC00206=459544
BC00207=459544
BC00208=459544
BC00209=459540
BC00210=533216
BC00211=533216
BC00212=492150
BC00213=423885
BC00214=423885
BC00215=423885
BC00216=423885
BC00217=423885
BC00218=493160
BC00219=493160
BC00220=493160
BC00221=493160
BC00222=493160
BC00223=493160
BC00224=539180
BC00225=539180
BC00226=539180
BC00227=539180
BC00228=539180
BC00229=539180
BC00230=525487
BC00231=485388
BC00232=485386
BC00233=485384
BC00234=485384
BC00235=485384
BC00236=485384
BC00237=485384
BC00238=485384
BC00239=485384
BC00240=485384
BC00241=635507
BC00242=635507
BC00243=635507
BC00244=635509
BC00245=635509
BC00246=635509
BC00247=635509
BC00248=635509
BC00249=603035
BC00250=594948
BC00251=594948
BC00252=594948
BC00253=594948
BC00254=594948
BC00255=594948
BC00256=594948
BC00257=600591
BC00258=600589
BC00259=600589
BC00260=600589
BC00261=600589
BC00262=600589
BC00263=600589
BC00264=623637
BC00265=623637
BC00266=623637
BC00267=623637
BC00268=623637
BC00269=623637
BC00270=623637
BC00271=623637
BC00272=623637
BC00273=623637
BC00274=623637
BC00275=623637
BC00276=623637
BC00277=623637
BC00278=623637
BC00279=758391
BC00280=758391
BC00281=758391
BC00282=758391
BC00283=758391
BC00284=758391
BC00285=758391
BC00286=758391
BC00287=758391
BC00288=669704
BC00289=669704
BC00290=669706
BC00291=669704
BC00292=669704
BC00293=669704
BC00294=784942
BC00295=784942
BC00296=784942
BC00297=784942
BC00298=784942
BC00299=784942
BC00300=807985
BC00301=807985
BC00302=807985
BC00303=807985
BC00304=807985
BC00305=807985
BC00306=807985
BC00307=784942
BC00308=784942
BC00309=784942
BC00310=784942
BC00311=784942
BC00312=784942
BC00313=784942
BC00314=784942
BC00315=785203
BC00316=785203
BC00317=785203
BC00318=895226
BC00319=895226
BC00320=895226
BC00321=895226
BC00322=895226
BC00323=895226
BC00324=895226
BC00325=895226
BC00326=895226
BC00327=895226
BC00328=906894
BC00329=906894
BC00330=963281
BC00331=963281
BC00332=963281
BC00333=969297
BC00334=969297
BC00335=969297
BC00336=969297
BC00337=969297
BC00338=969297
BC00339=969297
BC00340=969297
BC00341=969297
BC00342=969297
BC00343=969297
BC00344=969297
BC00345=927243
BC00346=883644
BC00347=475149
BC00348=445130
BC00349=445130
BC00350=445130
BC00351=445130
BC00352=445130
BC00353=445710
BC00354=445126
BC00355=445722
BC00356=484130
BC00357=492177
BC00358=481766
BC00359=492273
BC00360=473247
BC00361=480563
BC00362=473247
BC00363=480984
BC00364=519338
BC00365=527043
BC00366=519335
BC00367=519335
BC00368=550079
BC00369=550079
BC00370=542403
BC00371=542207
BC00372=542207
BC00373=542207
BC00374=542207
BC00375=542207
BC00376=492150
BC00377=423885
BC00378=471005
BC00379=487965
BC00380=477405
BC00381=472948
BC00382=455020
BC00383=453643
BC00384=453643
BC00385=493160
BC00386=521199
BC00387=521199
BC00388=521199
BC00389=521199
BC00390=484684
BC00391=484684
BC00392=484684
BC00393=484684
BC00394=484684
BC00395=484684
BC00396=484684
BC00397=493160
BC00398=582810
BC00399=655182
BC00400=655182
BC00401=655182
BC00402=655182
BC00403=716328
BC00404=716642
BC00405=582810
BC00406=493160
BC00407=542207
BC00408=542207
BC00409=542207
BC00410=590944
BC00411=557139
BC00412=543764
BC00413=551223
BC00414=543862
BC00415=551454
BC00416=589824
BC00417=589880
BC00418=589882
BC00419=589824
BC00420=612873
BC00421=620543
BC00422=613014
BC00423=612873
BC00424=612873
BC00425=584417
BC00426=584417
BC00427=584417
BC00428=584417
BC00429=584417
BC00430=590475
BC00431=610524
BC00432=594969
BC00433=594969
BC00434=594969
BC00435=593583
BC00436=552811
BC00437=552811
BC00438=552811
BC00439=552811
BC00440=612529
BC00441=612529
BC00442=620193
BC00443=620193
BC00444=620193
BC00445=620193
BC00446=620193
BC00447=620193
BC00448=620193
BC00449=812803
BC00450=887783
BC00451=897274
BC00452=900756
BC00453=962030
BC00454=962387
BC00455=853059
BC00456=542207
BC00457=542207
BC00458=542207
BC00459=542207
BC00460=574221
BC00461=593265
BC00462=593265
BC00463=612873
BC00464=618023
BC00465=625391
BC00466=633099
BC00467=633139
BC00468=664106
BC00469=671474
BC00470=679182
BC00471=679222
BC00472=633159
BC00473=633159
BC00474=633159
BC00475=681733
BC00476=681733
BC00477=740703
BC00478=740703
BC00479=740703
BC00480=740703
BC00481=743159
BC00482=735397
BC00483=733039
BC00484=733103
BC00485=748464
BC00486=748464
BC00487=748464
BC00488=748464
BC00489=748464
BC00490=748464
BC00491=620193
BC00492=626283
BC00493=635598
BC00494=635765
BC00495=635816
BC00496=643271
BC00497=641590
BC00498=641590
BC00499=685792
BC00500=685797
BC00501=685792
BC00502=685792
BC00503=685792
BC00504=771083
BC00505=750783
BC00506=758455
BC00507=750783
BC00508=750783
BC00509=719658
BC00510=685920
BC00511=620193
BC00512=620193
BC00513=561542
BC00514=498768
BC00515=407896
BC00516=407892
BC00517=469047
BC00518=469397
BC00519=524165
BC00520=524165
BC00521=733103
BC00522=733103
BC00523=733103
BC00524=756144
BC00525=756144
BC00526=756144
BC00527=771424
BC00528=771424
BC00529=779179
BC00530=771424
BC00531=794504
BC00532=794504
BC00533=801218
BC00534=794504
BC00535=840598
BC00536=840598
BC00537=846974
BC00538=840598
BC00539=840598
BC00540=840598
BC00541=840598
BC00542=840598
BC00543=795297
BC00544=741582
BC00545=733102
BC00546=620193
BC00547=700154
BC00548=704277
BC00549=716233
BC00550=716233
BC00551=716233
BC00552=716233
BC00553=716233
BC00554=733710
BC00555=733710
BC00556=733710
BC00557=733710
BC00558=742336
BC00559=742336
BC00560=742336
BC00561=763798
BC00562=742336
BC00563=742336
BC00564=742336
BC00565=742336
BC00566=743633
BC00567=750104
BC00568=672725
BC00569=672725
BC00570=672725
BC00571=576077
BC00572=465158
BC00573=407896
BC00574=407896
BC00575=407896
BC00576=407896
BC00577=407896
BC00578=407896
BC00579=471446
BC00580=524165
BC00581=524165
BC00582=733103
BC00583=733103
BC00584=733103
BC00585=756144
BC00586=756144
BC00587=756144
BC00588=846020
BC00589=846020
BC00590=853267
BC00591=846020
BC00592=869044
BC00593=869046
BC00594=876239
BC00595=869044
BC00596=869044
BC00597=868629
BC00598=860147
BC00599=840598
BC00600=840598
BC00601=795297
BC00602=733103
BC00603=733103
BC00604=762701
BC00605=816902
BC00606=816902
BC00607=837114
BC00608=816902
BC00609=816839
BC00610=816869
BC00611=816900
BC00612=816902
BC00613=816839
BC00614=816902
BC00615=837114
BC00616=903552
BC00617=903552
BC00618=897057
BC00619=903398
BC00620=903552
BC00621=903552
BC00622=903552
BC00623=903552
BC00624=903552
BC00625=903552
BC00626=903552
BC00627=848113
BC00628=815298
BC00629=672725
BC00630=672725
BC00631=672725
BC00632=576077
BC00633=513681
BC00634=534857
BC00635=557970
BC00636=557452
BC00637=618309
BC00638=618402
BC00639=618402
BC00640=618402
BC00641=618402
BC00642=733103
BC00643=748464
BC00644=957461
BC00645=939032
BC00646=955992
BC00647=946776
BC00648=1000598
BC00649=988507
BC00650=988507
BC00651=970092
BC00652=993094
BC00653=993094
BC00654=990114
BC00655=987237
BC00656=992538
BC00657=992538
BC00658=992538
BC00659=992538
BC00660=993094
BC00661=982648
BC00662=993094
BC00663=953359
BC00664=936837
BC00665=840598
BC00666=795297
BC00667=748875
BC00668=733103
BC00669=852584
BC00670=921533
BC00671=921533
BC00672=923427
BC00673=923499
BC00674=923499
BC00675=923501
BC00676=932594
BC00677=943380
BC00678=943380
BC00679=943380
BC00680=963295
BC00681=934184
BC00682=929661
BC00683=754884
BC00684=672725
BC00685=672725
BC00686=749842
BC00687=756681
BC00688=776639
BC00689=776639
BC00690=776639
BC00691=838373
BC00692=837995
BC00693=796760
BC00694=742282
///POSTYPE BASE
///RECTAN
///RCONF 0,0,0,0,0,0,0,0,0,0,0,0,0,0,0,0,0,0,0,0,0,0,0,0
P00006=-2.449,0.031,8.825,0.0000,0.0000,0.0000
P00058=0.000,0.000,3.000,0.0000,0.0000,0.0000
///RCONF 1,0,0,0,0,0,0,0,0,0,0,0,0,0,0,0,0,0,0,0,0,0,0,0
P00300=-0.036,-1.505,2.318,0.0000,0.0000,0.0000
///RCONF 0,0,0,0,0,0,0,0,0,0,0,0,0,0,0,0,0,0,0,0,0,0,0,0
P00301=0.005,-4.708,-4.628,0.0000,0.0000,0.0000
P00302=0.052,-2.937,-4.426,0.0000,0.0000,0.0000
P00303=-0.004,-1.437,-4.584,0.0000,0.0000,0.0000
P00304=0.028,-1.666,-4.234,0.0000,0.0000,0.0000
P00305=-0.003,-1.920,-3.501,0.0000,0.0000,0.0000
P00306=0.015,-2.252,-3.054,0.0000,0.0000,0.0000
P00307=0.019,-2.151,-5.077,0.0000,0.0000,0.0000
P00308=-0.003,-2.092,-4.888,0.0000,0.0000,0.0000
P00309=-0.040,-2.205,-4.992,0.0000,0.0000,0.0000
P00310=-0.006,-2.490,-5.925,0.0000,0.0000,0.0000
P00311=-0.007,-2.079,-5.307,0.0000,0.0000,0.0000
P00312=-0.032,2.202,-7.632,0.0000,0.0000,0.0000
///RCONF 1,0,0,0,0,0,0,0,0,0,0,0,0,0,0,0,0,0,0,0,0,0,0,0
P00313=-0.088,1.055,2.110,0.0000,0.0000,0.0000
P00314=-0.055,1.752,1.634,0.0000,0.0000,0.0000
P00315=-0.074,0.897,1.645,0.0000,0.0000,0.0000
P00316=0.009,2.112,2.075,0.0000,0.0000,0.0000
P00317=-0.015,2.781,3.126,0.0000,0.0000,0.0000
P00318=-0.086,2.132,2.037,0.0000,0.0000,0.0000
///RCONF 0,0,0,0,0,0,0,0,0,0,0,0,0,0,0,0,0,0,0,0,0,0,0,0
P00350=11.519,-0.008,1.149,0.0000,0.0000,0.0000
P00351=13.563,-0.027,-0.653,0.0000,0.0000,0.0000
P00352=13.252,-0.027,-0.827,0.0000,0.0000,0.0000
P00353=10.971,-0.082,0.776,0.0000,0.0000,0.0000
P00354=-0.024,2.508,-1.824,0.0000,0.0000,0.0000
P00355=-0.001,2.528,-1.131,0.0000,0.0000,0.0000
P00356=-0.034,2.921,-0.262,0.0000,0.0000,0.0000
P00357=0.003,3.386,-0.091,0.0000,0.0000,0.0000
P00358=0.014,3.037,-0.020,0.0000,0.0000,0.0000
P00359=-0.005,2.731,0.912,0.0000,0.0000,0.0000
P00360=-0.011,3.412,0.438,0.0000,0.0000,0.0000
P00361=0.018,3.050,1.253,0.0000,0.0000,0.0000
P00401=3.430,-0.021,1.131,0.0000,0.0000,0.0000
P00402=-0.253,1.107,3.062,0.0000,0.0000,0.0000
P00403=-3.666,-0.015,5.328,0.0000,0.0000,0.0000
///RCONF 1,0,0,0,0,0,0,0,0,0,0,0,0,0,0,0,0,0,0,0,0,0,0,0
P00404=0.029,4.189,-1.030,0.0000,0.0000,0.0000
///RCONF 0,0,0,0,0,0,0,0,0,0,0,0,0,0,0,0,0,0,0,0,0,0,0,0
P00405=2.420,0.007,1.427,0.0000,0.0000,0.0000
P00406=3.513,-0.022,0.429,0.0000,0.0000,0.0000
///RCONF 1,0,0,0,1,0,0,0,0,0,0,0,0,0,0,0,0,0,0,0,0,0,0,0
P00407=-0.029,2.348,-1.469,0.0000,0.0000,0.0000
P00408=0.010,1.346,-1.479,0.0000,0.0000,0.0000
///RCONF 1,0,0,0,0,0,0,0,0,0,0,0,0,0,0,0,0,0,0,0,0,0,0,0
P00409=-0.026,2.090,-1.483,0.0000,0.0000,0.0000
P00410=0.001,4.491,-0.583,0.0000,0.0000,0.0000
///RCONF 1,0,0,0,1,0,0,0,0,0,0,0,0,0,0,0,0,0,0,0,0,0,0,0
P00411=-0.015,3.627,0.872,0.0000,0.0000,0.0000
P00412=0.002,3.829,0.787,0.0000,0.0000,0.0000
P00413=0.046,0.107,-0.040,0.0000,0.0000,0.0000
///RCONF 1,0,0,0,0,0,0,0,0,0,0,0,0,0,0,0,0,0,0,0,0,0,0,0
P00414=0.046,0.800,0.739,0.0000,0.0000,0.0000
///RCONF 0,0,0,0,0,0,0,0,0,0,0,0,0,0,0,0,0,0,0,0,0,0,0,0
P00415=-1.781,-1.303,3.250,0.0000,0.0000,0.0000
P00416=0.027,1.119,3.078,0.0000,0.0000,0.0000
///RCONF 1,0,0,0,1,0,0,0,0,0,0,0,0,0,0,0,0,0,0,0,0,0,0,0
P00417=0.059,4.721,3.973,0.0000,0.0000,0.0000
//INST
///DATE 2024/10/28 15:05
///ATTR SC,RW
///GROUP1 RB1,BS1
NOP
CALL JOB:MOVE_INTO_TUNNEL
MOVJ C00000 BC00000 VJ=50.00
MOVJ C00001 BC00001 VJ=40.00
MOVJ C00002 BC00002 VJ=40.00
MOVL C00003 BC00003 V=666.7
MOVJ C00004 BC00004 VJ=30.00
MOVL C00005 BC00005 V=500.0
'------------------------
'W31.2
'------------------------
MOVL C00006 BC00006 V=166.7 PL=0
REFP 3 C00007 BC00007
CALL JOB:SEARCH-R1
SET P0300 P0006
SFTON P0300
MOVL C00008 BC00008 V=166.7 PL=0
REFP 3 C00009 BC00009
CALL JOB:SEARCH-R1
SET P0300 P0006
SFTON P0300
MOVL C00010 BC00010 V=166.7 PL=0
SFTOF
'------------------------
'W31.4
'------------------------
MOVL C00011 BC00011 V=500.0
MOVL C00012 BC00012 V=166.7 PL=0
REFP 3 C00013 BC00013
CALL JOB:SEARCH-R1
SET P0301 P0006
SFTON P0301
MOVL C00014 BC00014 V=166.7 PL=0
REFP 3 C00015 BC00015
CALL JOB:SEARCH-R1
SET P0301 P0006
SFTON P0301
MOVL C00016 BC00016 V=166.7 PL=0
SFTOF
'------------------------
'W31.6
'------------------------
MOVL C00017 BC00017 V=500.0
MOVL C00018 BC00018 V=166.7 PL=0
REFP 3 C00019 BC00019
CALL JOB:SEARCH-R1
SET P0302 P0006
SFTON P0302
MOVL C00020 BC00020 V=166.7 PL=0
REFP 3 C00021 BC00021
CALL JOB:SEARCH-R1
SET P0302 P0006
SFTON P0302
MOVL C00022 BC00022 V=166.7 PL=0
SFTOF
'------------------------
'W31.8
'------------------------
MOVL C00023 BC00023 V=500.0
MOVL C00024 BC00024 V=166.7 PL=0
REFP 3 C00025 BC00025
CALL JOB:SEARCH-R1
SET P0303 P0006
SFTON P0303
MOVL C00026 BC00026 V=166.7 PL=0
REFP 3 C00027 BC00027
CALL JOB:SEARCH-R1
SET P0303 P0006
SFTON P0303
MOVL C00028 BC00028 V=166.7 PL=0
SFTOF
'------------------------
'W31.9
'------------------------
MOVL C00029 BC00029 V=500.0
MOVL C00030 BC00030 V=166.7 PL=0
REFP 3 C00031 BC00031
CALL JOB:SEARCH-R1
SET P0304 P0006
SFTON P0304
MOVL C00032 BC00032 V=166.7 PL=0
REFP 3 C00033 BC00033
CALL JOB:SEARCH-R1
SET P0304 P0006
SFTON P0304
MOVL C00034 BC00034 V=166.7 PL=0
SFTOF
'------------------------
'W31.11
'------------------------
MOVL C00035 BC00035 V=500.0
MOVL C00036 BC00036 V=166.7 PL=0
REFP 3 C00037 BC00037
CALL JOB:SEARCH-R1
SET P0305 P0006
SFTON P0305
MOVL C00038 BC00038 V=166.7 PL=0
REFP 3 C00039 BC00039
CALL JOB:SEARCH-R1
SET P0305 P0006
SFTON P0305
MOVL C00040 BC00040 V=166.7 PL=0
SFTOF
'------------------------
'W31.13
'------------------------
MOVL C00041 BC00041 V=500.0
MOVL C00042 BC00042 V=166.7 PL=0
REFP 3 C00043 BC00043
CALL JOB:SEARCH-R1
SET P0306 P0006
SFTON P0306
MOVL C00044 BC00044 V=166.7 PL=0
REFP 3 C00045 BC00045
CALL JOB:SEARCH-R1
SET P0306 P0006
SFTON P0306
MOVL C00046 BC00046 V=166.7 PL=0
SFTOF
'------------------------
'W31.14
'------------------------
MOVL C00047 BC00047 V=500.0
MOVL C00048 BC00048 V=166.7 PL=0
REFP 3 C00049 BC00049
CALL JOB:SEARCH-R1
SET P0307 P0006
SFTON P0307
MOVL C00050 BC00050 V=166.7 PL=0
REFP 3 C00051 BC00051
CALL JOB:SEARCH-R1
SET P0307 P0006
SFTON P0307
MOVL C00052 BC00052 V=166.7 PL=0
SFTOF
'------------------------
'W31.16
'------------------------
MOVL C00053 BC00053 V=500.0
MOVL C00054 BC00054 V=166.7 PL=0
REFP 3 C00055 BC00055
CALL JOB:SEARCH-R1
SET P0308 P0006
SFTON P0308
MOVL C00056 BC00056 V=166.7 PL=0
REFP 3 C00057 BC00057
CALL JOB:SEARCH-R1
SET P0308 P0006
SFTON P0308
MOVL C00058 BC00058 V=166.7 PL=0
SFTOF
MOVL C00059 BC00059 V=150.0
MOVL C00060 BC00060 V=333.3
MOVL C00061 BC00061 V=500.0
MOVL C00062 BC00062 V=500.0
MOVJ C00063 BC00063 VJ=50.00
MOVL C00064 BC00064 V=666.7
MOVL C00065 BC00065 V=500.0
MOVL C00066 BC00066 V=333.3
'------------------------
'W31.18
'------------------------
MOVL C00067 BC00067 V=166.7
MOVL C00068 BC00068 V=133.3 PL=0
REFP 3 C00069 BC00069
CALL JOB:SEARCH-R1
SET P0309 P0006
SFTON P0309
MOVL C00070 BC00070 V=66.7 PL=0
REFP 3 C00071 BC00071
CALL JOB:SEARCH-R1
SET P0309 P0006
SFTON P0309
MOVL C00072 BC00072 V=66.7 PL=0
SFTOF
'------------------------
'W31.19
'------------------------
MOVL C00073 BC00073 V=500.0
MOVL C00074 BC00074 V=166.7 PL=0
REFP 3 C00075 BC00075
CALL JOB:SEARCH-R1
SET P0310 P0006
SFTON P0310
MOVL C00076 BC00076 V=166.7 PL=0
REFP 3 C00077 BC00077
CALL JOB:SEARCH-R1
SET P0310 P0006
SFTON P0310
MOVL C00078 BC00078 V=166.7 PL=0
SFTOF
'------------------------
'W31.21
'------------------------
MOVL C00079 BC00079 V=500.0
MOVL C00080 BC00080 V=166.7 PL=0
REFP 3 C00081 BC00081
CALL JOB:SEARCH-R1
SET P0311 P0006
SFTON P0311
MOVL C00082 BC00082 V=166.7 PL=0
REFP 3 C00083 BC00083
CALL JOB:SEARCH-R1
SET P0311 P0006
SFTON P0311
MOVL C00084 BC00084 V=166.7 PL=0
SFTOF
'------------------------
'W31.22
'------------------------
MOVL C00085 BC00085 V=500.0
MOVL C00086 BC00086 V=166.7 PL=0
REFP 3 C00087 BC00087
CALL JOB:SEARCH-R1
SET P0312 P0006
SFTON P0312
MOVL C00088 BC00088 V=166.7 PL=0
REFP 3 C00089 BC00089
CALL JOB:SEARCH-R1
SET P0312 P0006
SFTON P0312
MOVL C00090 BC00090 V=166.7 PL=0
SFTOF
'------------------------
'W31.24
'------------------------
MOVL C00091 BC00091 V=500.0
MOVL C00092 BC00092 V=166.7 PL=0
REFP 3 C00093 BC00093
CALL JOB:SEARCH-R1
SET P0313 P0006
SFTON P0313
MOVL C00094 BC00094 V=166.7 PL=0
REFP 3 C00095 BC00095
CALL JOB:SEARCH-R1
SET P0313 P0006
SFTON P0313
MOVL C00096 BC00096 V=166.7 PL=0
SFTOF
'------------------------
'W31.26
'------------------------
MOVL C00097 BC00097 V=500.0
MOVL C00098 BC00098 V=166.7 PL=0
REFP 3 C00099 BC00099
CALL JOB:SEARCH-R1
SET P0314 P0006
SFTON P0314
MOVL C00100 BC00100 V=166.7 PL=0
REFP 3 C00101 BC00101
CALL JOB:SEARCH-R1
SET P0314 P0006
SFTON P0314
MOVL C00102 BC00102 V=166.7 PL=0
SFTOF
'------------------------
'W31.27
'------------------------
MOVL C00103 BC00103 V=500.0
MOVL C00104 BC00104 V=166.7 PL=0
REFP 3 C00105 BC00105
CALL JOB:SEARCH-R1
SET P0315 P0006
SFTON P0315
MOVL C00106 BC00106 V=166.7 PL=0
REFP 3 C00107 BC00107
CALL JOB:SEARCH-R1
SET P0315 P0006
SFTON P0315
MOVL C00108 BC00108 V=166.7 PL=0
SFTOF
'------------------------
'W31.29
'------------------------
MOVL C00109 BC00109 V=500.0
MOVL C00110 BC00110 V=166.7 PL=0
REFP 3 C00111 BC00111
CALL JOB:SEARCH-R1
SET P0316 P0006
SFTON P0316
MOVL C00112 BC00112 V=166.7 PL=0
REFP 3 C00113 BC00113
CALL JOB:SEARCH-R1
SET P0316 P0006
SFTON P0316
MOVL C00114 BC00114 V=166.7 PL=0
SFTOF
MOVL C00115 BC00115 V=333.3
MOVL C00116 BC00116 V=666.7
MOVL C00117 BC00117 V=666.7
MOVL C00118 BC00118 V=666.7
MOVL C00119 BC00119 V=666.7
MOVL C00120 BC00120 V=666.7
MOVL C00121 BC00121 V=666.7
MOVL C00122 BC00122 V=333.3
MOVL C00123 BC00123 V=250.0
'------------------------
'W31.31
'------------------------
MOVL C00124 BC00124 V=500.0
MOVL C00125 BC00125 V=166.7 PL=0
REFP 3 C00126 BC00126
CALL JOB:SEARCH-R1
SET P0317 P0006
SFTON P0317
MOVL C00127 BC00127 V=166.7 PL=0
REFP 3 C00128 BC00128
CALL JOB:SEARCH-R1
SET P0317 P0006
SFTON P0317
MOVL C00129 BC00129 V=166.7 PL=0
SFTOF
'------------------------
'W31.32
'------------------------
MOVL C00130 BC00130 V=250.0
MOVL C00131 BC00131 V=166.7 PL=0
REFP 3 C00132 BC00132
CALL JOB:SEARCH-R1
SET P0318 P0006
SFTON P0318
MOVL C00133 BC00133 V=166.7 PL=0
REFP 3 C00134 BC00134
CALL JOB:SEARCH-R1
SET P0318 P0006
SFTON P0318
MOVL C00135 BC00135 V=166.7 PL=0
SFTOF
MOVL C00136 BC00136 V=250.0
MOVL C00137 BC00137 V=333.3
MOVL C00138 BC00138 V=333.3
MOVL C00139 BC00139 V=666.7
MOVJ C00140 BC00140 VJ=50.00
MOVJ C00141 BC00141 VJ=50.00
MOVJ C00142 BC00142 VJ=50.00
MOVJ C00143 BC00143 VJ=10.00
MOVJ C00144 BC00144 VJ=50.00
MOVJ C00145 BC00145 VJ=50.00
MOVJ C00146 BC00146 VJ=30.00
MOVL C00147 BC00147 V=166.7
'------------------------
'W214B L
'------------------------
MOVL C00148 BC00148 V=166.7 PL=0
REFP 3 C00149 BC00149
CALL JOB:SEARCH-R1
IMOV P0058 V=16.7
SET P0350 P0006
SFTON P0350
REFP 3 C00150 BC00150
CALL JOB:SEARCH-R1
SET P0350 P0006
SFTON P0350
MOVL C00151 BC00151 V=166.7 PL=0
SFTOF
'------------------------
'W214A P
'------------------------
MOVJ C00152 BC00152 VJ=40.00
MOVL C00153 BC00153 V=166.7 PL=0
REFP 3 C00154 BC00154
CALL JOB:SEARCH-R1
IMOV P0058 V=16.7
SET P0351 P0006
SFTON P0351
REFP 3 C00155 BC00155
CALL JOB:SEARCH-R1
SET P0351 P0006
SFTON P0351
MOVL C00156 BC00156 V=166.7 PL=0
SFTOF
'------------------------
'W219B L
'------------------------
MOVJ C00157 BC00157 VJ=40.00
MOVL C00158 BC00158 V=166.7 PL=0
REFP 3 C00159 BC00159
CALL JOB:SEARCH-R1
IMOV P0058 V=16.7
SET P0352 P0006
SFTON P0352
REFP 3 C00160 BC00160
CALL JOB:SEARCH-R1
SET P0352 P0006
SFTON P0352
MOVL C00161 BC00161 V=166.7 PL=0
SFTOF
'------------------------
'W219B P
'------------------------
MOVJ C00162 BC00162 VJ=40.00
MOVL C00163 BC00163 V=166.7 PL=0
REFP 3 C00164 BC00164
CALL JOB:SEARCH-R1
IMOV P0058 V=16.7
SET P0353 P0006
SFTON P0353
REFP 3 C00165 BC00165
CALL JOB:SEARCH-R1
SET P0353 P0006
SFTON P0353
MOVL C00166 BC00166 V=166.7 PL=0
SFTOF
'------------------------
'W213B L
'------------------------
MOVJ C00167 BC00167 VJ=40.00
MOVL C00168 BC00168 V=166.7 PL=0
REFP 3 C00169 BC00169
CALL JOB:SEARCH-R1
IMOV P0058 V=16.7
SET P0354 P0006
SFTON P0354
REFP 3 C00170 BC00170
CALL JOB:SEARCH-R1
SET P0354 P0006
SFTON P0354
MOVL C00171 BC00171 V=166.7 PL=0
SFTOF
'------------------------
'W213B P
'------------------------
MOVJ C00172 BC00172 VJ=40.00
MOVL C00173 BC00173 V=166.7 PL=0
REFP 3 C00174 BC00174
CALL JOB:SEARCH-R1
IMOV P0058 V=16.7
SET P0355 P0006
SFTON P0355
REFP 3 C00175 BC00175
CALL JOB:SEARCH-R1
SET P0355 P0006
SFTON P0355
MOVL C00176 BC00176 V=166.7 PL=0
SFTOF
'------------------------
'W218B L
'------------------------
MOVJ C00177 BC00177 VJ=40.00
MOVL C00178 BC00178 V=166.7 PL=0
REFP 3 C00179 BC00179
CALL JOB:SEARCH-R1
IMOV P0058 V=16.7
SET P0356 P0006
SFTON P0356
REFP 3 C00180 BC00180
CALL JOB:SEARCH-R1
SET P0356 P0006
SFTON P0356
MOVL C00181 BC00181 V=166.7 PL=0
SFTOF
'------------------------
'W218B P
'------------------------
MOVJ C00182 BC00182 VJ=40.00
MOVL C00183 BC00183 V=166.7 PL=0
REFP 3 C00184 BC00184
CALL JOB:SEARCH-R1
IMOV P0058 V=16.7
SET P0357 P0006
SFTON P0357
REFP 3 C00185 BC00185
CALL JOB:SEARCH-R1
SET P0357 P0006
SFTON P0357
MOVL C00186 BC00186 V=166.7 PL=0
SFTOF
'------------------------
'W215B L
'------------------------
MOVJ C00187 BC00187 VJ=40.00
MOVL C00188 BC00188 V=166.7 PL=0
REFP 3 C00189 BC00189
CALL JOB:SEARCH-R1
IMOV P0058 V=16.7
SET P0358 P0006
SFTON P0358
REFP 3 C00190 BC00190
CALL JOB:SEARCH-R1
SET P0358 P0006
SFTON P0358
MOVL C00191 BC00191 V=166.7 PL=0
SFTOF
'------------------------
'W215B P
'------------------------
MOVL C00192 BC00192 V=666.7
MOVL C00193 BC00193 V=166.7 PL=0
REFP 3 C00194 BC00194
CALL JOB:SEARCH-R1
IMOV P0058 V=16.7
SET P0359 P0006
SFTON P0359
REFP 3 C00195 BC00195
CALL JOB:SEARCH-R1
SET P0359 P0006
SFTON P0359
MOVL C00196 BC00196 V=166.7 PL=0
SFTOF
'------------------------
'W217B L
'------------------------
MOVL C00197 BC00197 V=666.7
MOVL C00198 BC00198 V=166.7 PL=0
REFP 3 C00199 BC00199
CALL JOB:SEARCH-R1
IMOV P0058 V=16.7
SET P0360 P0006
SFTON P0360
REFP 3 C00200 BC00200
CALL JOB:SEARCH-R1
SET P0360 P0006
SFTON P0360
MOVL C00201 BC00201 V=166.7 PL=0
SFTOF
'------------------------
'W217B P
'------------------------
MOVL C00202 BC00202 V=666.7
MOVL C00203 BC00203 V=166.7 PL=0
REFP 3 C00204 BC00204
CALL JOB:SEARCH-R1
IMOV P0058 V=16.7
SET P0361 P0006
SFTON P0361
REFP 3 C00205 BC00205
CALL JOB:SEARCH-R1
SET P0361 P0006
SFTON P0361
MOVL C00206 BC00206 V=166.7 PL=0
SFTOF
MOVL C00207 BC00207 V=333.3
MOVL C00208 BC00208 V=666.7
MOVL C00209 BC00209 V=666.7
MOVJ C00210 BC00210 VJ=50.00
MOVJ C00211 BC00211 VJ=50.00
COMM MOVJ C00212 BC00212 VJ=40.00
COMM MOVJ C00213 BC00213 VJ=40.00
COMM MOVJ C00214 BC00214 VJ=25.00
COMM MOVJ C00215 BC00215 VJ=30.00
COMM MOVJ C00216 BC00216 VJ=30.00
COMM MOVJ C00217 BC00217 VJ=20.00
COMM MOVL C00218 BC00218 V=500.0
COMM '------------------------
COMM 'W27.4
COMM '------------------------
COMM MOVL C00219 BC00219 V=166.7 PL=0
COMM REFP 3 C00220 BC00220
COMM CALL JOB:SEARCH-R1
COMM SET P0401 P0006
COMM SFTON P0401
COMM MOVL C00221 BC00221 V=166.7 PL=0
COMM REFP 3 C00222 BC00222
COMM CALL JOB:SEARCH-R1
COMM SET P0401 P0006
COMM SFTON P0401
COMM MOVL C00223 BC00223 V=166.7 PL=0
COMM SFTOF
COMM '------------------------
COMM 'W27.6
COMM '------------------------
COMM MOVL C00224 BC00224 V=666.7
COMM MOVL C00225 BC00225 V=166.7 PL=0
COMM REFP 3 C00226 BC00226
COMM CALL JOB:SEARCH-R1
COMM SET P0402 P0006
COMM SFTON P0402
COMM MOVL C00227 BC00227 V=166.7 PL=0
COMM REFP 3 C00228 BC00228
COMM CALL JOB:SEARCH-R1
COMM SET P0402 P0006
COMM SFTON P0402
COMM MOVL C00229 BC00229 V=166.7 PL=0
COMM SFTOF
COMM MOVL C00230 BC00230 V=500.0
COMM MOVL C00231 BC00231 V=500.0
COMM '------------------------
COMM 'W27.8
COMM '------------------------
COMM MOVL C00232 BC00232 V=333.3
COMM MOVL C00233 BC00233 V=166.7 PL=0
COMM REFP 3 C00234 BC00234
COMM CALL JOB:SEARCH-R1
COMM SET P0403 P0006
COMM SFTON P0403
COMM MOVL C00235 BC00235 V=166.7 PL=0
COMM REFP 3 C00236 BC00236
COMM CALL JOB:SEARCH-R1
COMM SET P0403 P0006
COMM SFTON P0403
COMM MOVL C00237 BC00237 V=166.7 PL=0
COMM SFTOF
COMM MOVJ C00238 BC00238 VJ=25.00
COMM MOVJ C00239 BC00239 VJ=25.00
COMM MOVJ C00240 BC00240 VJ=30.00
COMM MOVJ C00241 BC00241 VJ=40.00
COMM MOVJ C00242 BC00242 VJ=30.00
COMM '------------------------
COMM 'W27.9
COMM '------------------------
COMM MOVL C00243 BC00243 V=500.0
COMM MOVL C00244 BC00244 V=166.7 PL=0
COMM REFP 3 C00245 BC00245
COMM CALL JOB:SEARCH-R1
COMM SET P0404 P0006
COMM SFTON P0404
COMM MOVL C00246 BC00246 V=166.7 PL=0
COMM REFP 3 C00247 BC00247
COMM CALL JOB:SEARCH-R1
COMM SET P0404 P0006
COMM SFTON P0404
COMM MOVL C00248 BC00248 V=166.7 PL=0
COMM SFTOF
COMM MOVL C00249 BC00249 V=500.0
COMM '------------------------
COMM 'W27.11
COMM '------------------------
COMM MOVL C00250 BC00250 V=500.0
COMM MOVL C00251 BC00251 V=166.7 PL=0
COMM REFP 3 C00252 BC00252
COMM CALL JOB:SEARCH-R1
COMM SET P0405 P0006
COMM SFTON P0405
COMM MOVL C00253 BC00253 V=166.7 PL=0
COMM REFP 3 C00254 BC00254
COMM CALL JOB:SEARCH-R1
COMM SET P0405 P0006
COMM SFTON P0405
COMM MOVL C00255 BC00255 V=166.7 PL=0
COMM SFTOF
COMM MOVL C00256 BC00256 V=666.7
COMM MOVL C00257 BC00257 V=666.7
COMM '------------------------
COMM 'W27.13
COMM '------------------------
COMM MOVL C00258 BC00258 V=333.3
COMM MOVL C00259 BC00259 V=166.7 PL=0
COMM REFP 3 C00260 BC00260
COMM CALL JOB:SEARCH-R1
COMM SET P0406 P0006
COMM SFTON P0406
COMM MOVL C00261 BC00261 V=166.7 PL=0
COMM REFP 3 C00262 BC00262
COMM CALL JOB:SEARCH-R1
COMM SET P0406 P0006
COMM SFTON P0406
COMM MOVL C00263 BC00263 V=166.7 PL=0
COMM SFTOF
COMM '------------------------
COMM 'W27.14
COMM '------------------------
COMM MOVL C00264 BC00264 V=666.7
COMM MOVL C00265 BC00265 V=166.7 PL=0
COMM REFP 3 C00266 BC00266
COMM CALL JOB:SEARCH-R1
COMM SET P0407 P0006
COMM SFTON P0407
COMM MOVL C00267 BC00267 V=166.7 PL=0
COMM REFP 3 C00268 BC00268
COMM CALL JOB:SEARCH-R1
COMM SET P0407 P0006
COMM SFTON P0407
COMM MOVL C00269 BC00269 V=166.7 PL=0
COMM SFTOF
COMM MOVL C00270 BC00270 V=666.7
COMM '------------------------
COMM 'W27.16
COMM '------------------------
COMM MOVL C00271 BC00271 V=333.3
COMM MOVL C00272 BC00272 V=166.7 PL=0
COMM REFP 3 C00273 BC00273
COMM CALL JOB:SEARCH-R1
COMM SET P0408 P0006
COMM SFTON P0408
COMM MOVL C00274 BC00274 V=166.7 PL=0
COMM REFP 3 C00275 BC00275
COMM CALL JOB:SEARCH-R1
COMM SET P0408 P0006
COMM SFTON P0408
COMM MOVL C00276 BC00276 V=166.7 PL=0
COMM SFTOF
COMM MOVL C00277 BC00277 V=666.7
COMM MOVJ C00278 BC00278 VJ=30.00
COMM MOVJ C00279 BC00279 VJ=50.00
COMM MOVJ C00280 BC00280 VJ=40.00
COMM MOVJ C00281 BC00281 VJ=30.00
COMM '------------------------
COMM 'W27.18
COMM '------------------------
COMM MOVL C00282 BC00282 V=333.3
COMM MOVL C00283 BC00283 V=166.7 PL=0
COMM REFP 3 C00284 BC00284
COMM CALL JOB:SEARCH-R1
COMM SET P0409 P0006
COMM SFTON P0409
COMM MOVL C00285 BC00285 V=166.7 PL=0
COMM REFP 3 C00286 BC00286
COMM CALL JOB:SEARCH-R1
COMM SET P0409 P0006
COMM SFTON P0409
COMM MOVL C00287 BC00287 V=166.7 PL=0
COMM SFTOF
COMM '------------------------
COMM 'W27.19
COMM '------------------------
COMM MOVL C00288 BC00288 V=666.7
COMM MOVL C00289 BC00289 V=166.7 PL=0
COMM REFP 3 C00290 BC00290
COMM CALL JOB:SEARCH-R1
COMM SET P0410 P0006
COMM SFTON P0410
COMM MOVL C00291 BC00291 V=166.7 PL=0
COMM REFP 3 C00292 BC00292
COMM CALL JOB:SEARCH-R1
COMM SET P0410 P0006
COMM SFTON P0410
COMM MOVL C00293 BC00293 V=166.7 PL=0
COMM SFTOF
COMM MOVL C00294 BC00294 V=666.7
COMM '------------------------
COMM 'W27.21
COMM '------------------------
COMM MOVL C00295 BC00295 V=166.7 PL=0
COMM REFP 3 C00296 BC00296
COMM CALL JOB:SEARCH-R1
COMM SET P0411 P0006
COMM SFTON P0411
COMM MOVL C00297 BC00297 V=166.7 PL=0
COMM REFP 3 C00298 BC00298
COMM CALL JOB:SEARCH-R1
COMM SET P0411 P0006
COMM SFTON P0411
COMM MOVL C00299 BC00299 V=166.7 PL=0
COMM SFTOF
COMM '------------------------
COMM 'W27.22
COMM '------------------------
COMM MOVL C00300 BC00300 V=666.7
COMM MOVL C00301 BC00301 V=166.7 PL=0
COMM REFP 3 C00302 BC00302
COMM CALL JOB:SEARCH-R1
COMM SET P0412 P0006
COMM SFTON P0412
COMM MOVL C00303 BC00303 V=166.7 PL=0
COMM REFP 3 C00304 BC00304
COMM CALL JOB:SEARCH-R1
COMM SET P0412 P0006
COMM SFTON P0412
COMM MOVL C00305 BC00305 V=166.7 PL=0
COMM SFTOF
COMM MOVL C00306 BC00306 V=666.7
COMM MOVJ C00307 BC00307 VJ=30.00
COMM MOVL C00308 BC00308 V=500.0
COMM '------------------------
COMM 'W27.24
COMM '------------------------
COMM MOVL C00309 BC00309 V=666.7
COMM MOVL C00310 BC00310 V=166.7 PL=0
COMM REFP 3 C00311 BC00311
COMM CALL JOB:SEARCH-R1
COMM SET P0413 P0006
COMM SFTON P0413
COMM MOVL C00312 BC00312 V=166.7 PL=0
COMM REFP 3 C00313 BC00313
COMM CALL JOB:SEARCH-R1
COMM SET P0413 P0006
COMM SFTON P0413
COMM MOVL C00314 BC00314 V=166.7 PL=0
COMM SFTOF
COMM MOVL C00315 BC00315 V=666.7
COMM MOVJ C00316 BC00316 VJ=50.00
COMM MOVJ C00317 BC00317 VJ=50.00
COMM MOVJ C00318 BC00318 VJ=50.00
COMM MOVJ C00319 BC00319 VJ=20.00
COMM MOVJ C00320 BC00320 VJ=10.00
COMM '------------------------
COMM 'W27.26
COMM '------------------------
COMM MOVL C00321 BC00321 V=333.3
COMM MOVL C00322 BC00322 V=166.7 PL=0
COMM REFP 3 C00323 BC00323
COMM CALL JOB:SEARCH-R1
COMM SET P0414 P0006
COMM SFTON P0414
COMM MOVL C00324 BC00324 V=166.7 PL=0
COMM REFP 3 C00325 BC00325
COMM CALL JOB:SEARCH-R1
COMM SET P0414 P0006
COMM SFTON P0414
COMM MOVL C00326 BC00326 V=166.7 PL=0
COMM SFTOF
COMM MOVL C00327 BC00327 V=333.3
COMM MOVJ C00328 BC00328 VJ=30.00
COMM MOVJ C00329 BC00329 VJ=30.00
COMM MOVJ C00330 BC00330 VJ=30.00
COMM GETE D040 P0414 (1)
COMM GETE D041 P0414 (2)
COMM GETE D042 P0414 (3)
COMM SETE P0415 (1) D040
COMM SETE P0415 (2) D041
COMM SETE P0415 (3) D042
COMM '------------------------
COMM 'W27.29
COMM '------------------------
COMM MOVJ C00331 BC00331 VJ=30.00
COMM MOVJ C00332 BC00332 VJ=30.00
COMM MOVL C00333 BC00333 V=333.3
COMM MOVL C00334 BC00334 V=166.7 PL=0
COMM REFP 3 C00335 BC00335
COMM CALL JOB:SEARCH-R1
COMM SET P0416 P0006
COMM SFTON P0416
COMM MOVL C00336 BC00336 V=166.7 PL=0
COMM REFP 3 C00337 BC00337
COMM CALL JOB:SEARCH-R1
COMM SET P0416 P0006
COMM SFTON P0416
COMM MOVL C00338 BC00338 V=166.7 PL=0
COMM SFTOF
COMM '------------------------
COMM 'W27.31
COMM '------------------------
COMM MOVL C00339 BC00339 V=666.7
COMM MOVL C00340 BC00340 V=166.7 PL=0
COMM REFP 3 C00341 BC00341
COMM CALL JOB:SEARCH-R1
COMM SET P0417 P0006
COMM SFTON P0417
COMM MOVL C00342 BC00342 V=166.7 PL=0
COMM REFP 3 C00343 BC00343
COMM CALL JOB:SEARCH-R1
COMM SET P0417 P0006
COMM SFTON P0417
COMM MOVL C00344 BC00344 V=166.7 PL=0
COMM SFTOF
COMM '------------------------
COMM 'W27.32
COMM '------------------------
COMM MOVL C00345 BC00345 V=333.3
MOVJ C00346 BC00346 VJ=50.00
IFTHENEXP OT#(1457)=ON ANDEXP OT#(1441)=OFF
	 CALL JOB:TWIN_FRONT_SEARCH_-90ST-1_5340
ENDIF
IFTHENEXP OT#(1457)=OFF ANDEXP OT#(1441)=ON
	 CALL JOB:FRONT_SEARCH_-90ST-1_5340
ENDIF
MOVJ C00347 BC00347 VJ=50.00
MOVJ C00348 BC00348 VJ=50.00
MOVJ C00349 BC00349 VJ=50.00
MOVL C00350 BC00350 V=666.7
MOVJ C00351 BC00351 VJ=30.00
'------------------------
'W31.2
'------------------------
SFTON P0300
MOVL C00352 BC00352 V=333.3
MOVL C00353 BC00353 V=166.7 PL=0
MACRO1 MJ#(0) ARGF10
ARCON
MOVL C00354 BC00354 V=10.8
ARCOF
MOVL C00355 BC00355 V=166.7
SFTOF
'------------------------
'W31.4
'------------------------
SFTON P0301
MOVL C00356 BC00356 V=666.7
MOVL C00357 BC00357 V=166.7 PL=0
ARCON
MOVL C00358 BC00358 V=10.8
ARCOF
MOVL C00359 BC00359 V=166.7
SFTOF
'------------------------
'W31.6
'------------------------
SFTON P0302
MOVL C00360 BC00360 V=666.7
MOVL C00361 BC00361 V=166.7 PL=0
ARCON
MOVL C00362 BC00362 V=10.8
ARCOF
MOVL C00363 BC00363 V=166.7
SFTOF
'------------------------
'W31.8
'------------------------
SFTON P0303
MOVL C00364 BC00364 V=666.7
MOVL C00365 BC00365 V=166.7 PL=0
ARCON
MOVL C00366 BC00366 V=10.8
ARCOF
MOVL C00367 BC00367 V=166.7
SFTOF
'------------------------
'W31.9
'------------------------
SFTON P0304
MOVL C00368 BC00368 V=666.7
MOVL C00369 BC00369 V=166.7 PL=0
ARCON
MOVL C00370 BC00370 V=10.8
ARCOF
MOVL C00371 BC00371 V=166.7
SFTOF
MOVL C00372 BC00372 V=500.0
MOVL C00373 BC00373 V=500.0
MOVJ C00374 BC00374 VJ=50.00
MOVJ C00375 BC00375 VJ=50.00
COMM '::::::::::::::::::::::::::::::::
COMM '::::::::::::::::::::::::::::::::
COMM '::::::::::::::::::::::::::::::::
COMM '::::::::::::::::::::::::::::::::
COMM '::::::::::::::::::::::::::::::::
COMM MOVJ C00376 BC00376 VJ=40.00
COMM MOVJ C00377 BC00377 VJ=40.00
COMM MOVJ C00378 BC00378 VJ=40.00
COMM MOVJ C00379 BC00379 VJ=40.00
COMM MOVJ C00380 BC00380 VJ=40.00
COMM MOVJ C00381 BC00381 VJ=40.00
COMM '------------------------
COMM 'W27.2
COMM '------------------------
COMM MOVL C00382 BC00382 V=500.0
COMM SFTON P0401
COMM MOVL C00383 BC00383 V=166.7 PL=0
COMM MACRO1 MJ#(0) ARGF24
COMM ARCON
COMM MOVL C00384 BC00384 V=7.5
COMM ARCOF
COMM SFTOF
COMM 'BELKA PRZEJAZD
COMM MOVL C00385 BC00385 V=500.0
COMM '------------------------
COMM 'W27.6
COMM '------------------------
COMM SFTON P0402
COMM MOVL C00386 BC00386 V=500.0
COMM MOVL C00387 BC00387 V=166.7 PL=0
COMM MACRO1 MJ#(0) ARGF24
COMM ARCON
COMM MOVL C00388 BC00388 V=7.5
COMM ARCOF
COMM MOVL C00389 BC00389 V=166.7
COMM SFTOF
COMM MOVJ C00390 BC00390 VJ=20.00
COMM '------------------------
COMM 'W27.8
COMM '------------------------
COMM SFTON P0403
COMM MOVL C00391 BC00391 V=500.0
COMM MOVL C00392 BC00392 V=166.7 PL=0
COMM MACRO1 MJ#(0) ARGF24
COMM ARCON
COMM MOVL C00393 BC00393 V=7.5
COMM ARCOF
COMM MOVL C00394 BC00394 V=166.7
COMM SFTOF
COMM MOVL C00395 BC00395 V=500.0
COMM MOVJ C00396 BC00396 VJ=50.00
MOVJ C00397 BC00397 VJ=50.00
MOVJ C00398 BC00398 VJ=50.00
MOVJ C00399 BC00399 VJ=50.00
MOVL C00400 BC00400 V=666.7
'------------------------
'W213A
'------------------------
SFTON P0355
MOVL C00401 BC00401 V=666.7
MOVL C00402 BC00402 V=166.7 PL=0
MACRO1 MJ#(0) ARGF9
ARCON
SFTOF
SFTON P0354
MOVL C00403 BC00403 V=11.2
ARCOF
MOVL C00404 BC00404 V=333.3
SFTOF
MOVJ C00405 BC00405 VJ=50.00
MOVJ C00406 BC00406 VJ=50.00
MOVJ C00407 BC00407 VJ=50.00
MOVJ C00408 BC00408 VJ=50.00
MOVJ C00409 BC00409 VJ=30.00
MOVJ C00410 BC00410 VJ=20.00
MOVJ C00411 BC00411 VJ=20.00
'5.5.1
'------------------------
'W31.11
'------------------------
SFTON P0305
MOVL C00412 BC00412 V=333.3
MOVL C00413 BC00413 V=166.7 PL=0
MACRO1 MJ#(0) ARGF10
ARCON
MOVL C00414 BC00414 V=10.8
ARCOF
MOVL C00415 BC00415 V=166.7
SFTOF
'------------------------
'W31.13
'------------------------
SFTON P0306
MOVL C00416 BC00416 V=500.0
'SPR CZY W DOBRYM MIEJSCU SPOINA
MOVL C00417 BC00417 V=166.7 PL=0
ARCON
MOVL C00418 BC00418 V=10.8
ARCOF
MOVL C00419 BC00419 V=166.7
SFTOF
'------------------------
'W31.14
'------------------------
SFTON P0307
MOVL C00420 BC00420 V=333.3
MOVL C00421 BC00421 V=166.7 PL=0
ARCON
MOVL C00422 BC00422 V=8.3
ARCOF
MOVL C00423 BC00423 V=166.7
SFTOF
MOVL C00424 BC00424 V=333.3
MOVL C00425 BC00425 V=500.0
MOVJ C00426 BC00426 VJ=30.00
MOVJ C00427 BC00427 VJ=30.00
MOVJ C00428 BC00428 VJ=30.00
MOVJ C00429 BC00429 VJ=50.00
COMM '::::::::::::::::::::::::::::::::
COMM '::::::::::::::::::::::::::::::::
COMM '------------------------
COMM 'W27.9
COMM '------------------------
COMM '::::::::::::::::::::::::::::::::
COMM '::::::::::::::::::::::::::::::::
COMM MOVJ C00430 BC00430 VJ=25.00
COMM MOVJ C00431 BC00431 VJ=40.00
COMM SFTON P0404
COMM MOVL C00432 BC00432 V=500.0
COMM MOVL C00433 BC00433 V=166.7 PL=0
COMM MACRO1 MJ#(0) ARGF24
COMM ARCON
COMM MOVL C00434 BC00434 V=7.5
COMM ARCOF
COMM MOVL C00435 BC00435 V=166.7
COMM SFTOF
COMM '------------------------
COMM 'W27.11
COMM '------------------------
COMM SFTON P0406
COMM MOVL C00436 BC00436 V=666.7
COMM MOVL C00437 BC00437 V=166.7 PL=0
COMM MACRO1 MJ#(0) ARGF24
COMM ARCON
COMM MOVL C00438 BC00438 V=7.5
COMM ARCOF
COMM MOVL C00439 BC00439 V=166.7
COMM SFTOF
COMM '------------------------
COMM 'W27.13
'------------------------
COMM SFTON P0406
COMM MOVL C00440 BC00440 V=666.7
COMM MOVL C00441 BC00441 V=166.7 PL=0
COMM MACRO1 MJ#(0) ARGF24
COMM ARCON
COMM MOVL C00442 BC00442 V=7.5
COMM ARCOF
COMM MOVL C00443 BC00443 V=166.7
COMM SFTOF
COMM MOVJ C00444 BC00444 VJ=40.00
COMM MOVJ C00445 BC00445 VJ=50.00
COMM MOVJ C00446 BC00446 VJ=50.00
COMM MOVJ C00447 BC00447 VJ=50.00
MOVJ C00448 BC00448 VJ=50.00
'::::::::::::::::::::::::
'::::::::::::::::::::::::
'::::::::::::::::::::::::
'::::::::::::::::::::::::
'::::::::::::::::::::::::
'::::::::::::::::::::::::
'::::::::::::::::::::::::
MOVJ C00449 BC00449 VJ=50.00
MOVJ C00450 BC00450 VJ=50.00
'------------------------
'W214A
'------------------------
SFTON P0351
MOVL C00451 BC00451 V=500.0
MOVL C00452 BC00452 V=166.7 PL=0
MACRO1 MJ#(0) ARGF9
ARCON
SFTOF
SFTON P0350
MOVL C00453 BC00453 V=11.7
ARCOF
MOVL C00454 BC00454 V=333.3
SFTOF
MOVJ C00455 BC00455 VJ=50.00
MOVJ C00456 BC00456 VJ=50.00
MOVJ C00457 BC00457 VJ=50.00
MOVJ C00458 BC00458 VJ=40.00
MOVJ C00459 BC00459 VJ=50.00
MOVJ C00460 BC00460 VJ=30.00
MOVJ C00461 BC00461 VJ=30.00
MOVJ C00462 BC00462 VJ=30.00
MOVJ C00463 BC00463 VJ=30.00
'------------------------
'W31.16
'------------------------
SFTON P0308
MOVL C00464 BC00464 V=666.7
MOVL C00465 BC00465 V=166.7 PL=0
MACRO1 MJ#(0) ARGF10
ARCON
MOVL C00466 BC00466 V=10.8
ARCOF
MOVL C00467 BC00467 V=166.7
SFTOF
'------------------------
'W31.18
'------------------------
SFTON P0309
MOVL C00468 BC00468 V=666.7
MOVL C00469 BC00469 V=166.7 PL=0
MACRO1 MJ#(0) ARGF10
ARCON
MOVL C00470 BC00470 V=10.8
ARCOF
MOVL C00471 BC00471 V=166.7
SFTOF
MOVL C00472 BC00472 V=666.7
MOVL C00473 BC00473 V=666.7
MOVL C00474 BC00474 V=666.7
MOVL C00475 BC00475 V=833.3
MOVL C00476 BC00476 V=666.7
MOVL C00477 BC00477 V=666.7
MOVL C00478 BC00478 V=333.3
MOVL C00479 BC00479 V=333.3
MOVL C00480 BC00480 V=250.0
'------------------------
'W31.19
'------------------------
SFTON P0310
MOVL C00481 BC00481 V=333.3
MOVL C00482 BC00482 V=166.7 PL=0
ARCON
MOVL C00483 BC00483 V=10.8
ARCOF
MOVL C00484 BC00484 V=166.7
SFTOF
MOVL C00485 BC00485 V=333.3
MOVL C00486 BC00486 V=500.0
MOVL C00487 BC00487 V=666.7
MOVL C00488 BC00488 V=666.7
MOVJ C00489 BC00489 VJ=40.00
MOVJ C00490 BC00490 VJ=40.00
COMM '::::::::::::::::::::::::
COMM '::::::::::::::::::::::::
COMM '::::::::::::::::::::::::
COMM '::::::::::::::::::::::::
COMM '::::::::::::::::::::::::
COMM '::::::::::::::::::::::::
COMM '::::::::::::::::::::::::
COMM MOVJ C00491 BC00491 VJ=50.00
COMM MOVJ C00492 BC00492 VJ=30.00
COMM '::::::::::::::::::::::::::::::::
COMM '::::::::::::::::::::::::::::::::
COMM '------------------------
COMM 'W27.14
COMM '------------------------
COMM '::::::::::::::::::::::::::::::::
COMM '::::::::::::::::::::::::::::::::
COMM MOVL C00493 BC00493 V=500.0
COMM MOVL C00494 BC00494 V=500.0
COMM SFTON P0407
COMM MOVL C00495 BC00495 V=166.7 PL=0
COMM MACRO1 MJ#(0) ARGF24
COMM ARCON
COMM MOVL C00496 BC00496 V=7.5
COMM ARCOF
COMM MOVL C00497 BC00497 V=166.7
COMM SFTOF
COMM MOVJ C00498 BC00498 VJ=30.00
COMM '------------------------
COMM 'W27.16
COMM '------------------------
COMM SFTON P0408
COMM MOVL C00499 BC00499 V=500.0
COMM MOVL C00500 BC00500 V=166.7 PL=0
COMM MACRO1 MJ#(0) ARGF24
COMM ARCON
COMM MOVL C00501 BC00501 V=6.7
COMM ARCOF
COMM MOVL C00502 BC00502 V=166.7
COMM MOVL C00503 BC00503 V=666.7
COMM MOVJ C00504 BC00504 VJ=50.00
COMM SFTOF
COMM '------------------------
COMM 'W27.18
COMM '------------------------
COMM SFTON P0409
COMM MOVL C00505 BC00505 V=500.0
COMM MOVL C00506 BC00506 V=166.7 PL=0
COMM MACRO1 MJ#(0) ARGF24
COMM ARCON
COMM MOVL C00507 BC00507 V=7.5
COMM ARCOF
COMM MOVL C00508 BC00508 V=166.7
COMM SFTOF
COMM MOVJ C00509 BC00509 VJ=30.00
COMM MOVJ C00510 BC00510 VJ=30.00
COMM MOVJ C00511 BC00511 VJ=40.00
MOVJ C00512 BC00512 VJ=50.00
'::::::::::::::::::::::::
'::::::::::::::::::::::::
'::::::::::::::::::::::::
'::::::::::::::::::::::::
'::::::::::::::::::::::::
'::::::::::::::::::::::::
'::::::::::::::::::::::::
MOVJ C00513 BC00513 VJ=50.00
MOVJ C00514 BC00514 VJ=50.00
'------------------------
'W215A
'------------------------
SFTON P0359
MOVL C00515 BC00515 V=666.7
MOVL C00516 BC00516 V=166.7 PL=0
MACRO1 MJ#(0) ARGF9
ARCON
SFTOF
SFTON P0358
MOVL C00517 BC00517 V=11.7
ARCOF
MOVL C00518 BC00518 V=333.3
SFTOF
MOVJ C00519 BC00519 VJ=50.00
MOVJ C00520 BC00520 VJ=50.00
MOVJ C00521 BC00521 VJ=50.00
MOVJ C00522 BC00522 VJ=50.00
MOVJ C00523 BC00523 VJ=50.00
MOVJ C00524 BC00524 VJ=50.00
MOVJ C00525 BC00525 VJ=50.00
MOVL C00526 BC00526 V=500.0
'------------------------
'W31.21
'------------------------
SFTON P0311
MOVL C00527 BC00527 V=333.3
MOVL C00528 BC00528 V=166.7 PL=0
MACRO1 MJ#(0) ARGF10
ARCON
MOVL C00529 BC00529 V=10.8
ARCOF
MOVL C00530 BC00530 V=166.7
SFTOF
'------------------------
'W31.22
'------------------------
SFTON P0312
MOVL C00531 BC00531 V=666.7
MOVL C00532 BC00532 V=166.7 PL=0
ARCON
MOVL C00533 BC00533 V=10.8
ARCOF
MOVL C00534 BC00534 V=166.7
SFTOF
'------------------------
'W31.24
'------------------------
SFTON P0313
MOVL C00535 BC00535 V=666.7
MOVL C00536 BC00536 V=166.7 PL=0
ARCON
MOVL C00537 BC00537 V=10.8
ARCOF
MOVL C00538 BC00538 V=166.7
MOVL C00539 BC00539 V=166.7
MOVL C00540 BC00540 V=333.3
SFTOF
MOVL C00541 BC00541 V=333.3
MOVJ C00542 BC00542 VJ=30.00
MOVJ C00543 BC00543 VJ=30.00
MOVJ C00544 BC00544 VJ=50.00
MOVJ C00545 BC00545 VJ=50.00
COMM '::::::::::::::::::::::::
COMM '::::::::::::::::::::::::
COMM '::::::::::::::::::::::::
COMM '::::::::::::::::::::::::
COMM '::::::::::::::::::::::::
COMM '::::::::::::::::::::::::
COMM '::::::::::::::::::::::::
COMM MOVJ C00546 BC00546 VJ=50.00
COMM MOVJ C00547 BC00547 VJ=50.00
COMM '::::::::::::::::::::::::::::::::
COMM '::::::::::::::::::::::::::::::::
COMM '------------------------
COMM 'W27.19
COMM '------------------------
COMM '::::::::::::::::::::::::::::::::
COMM '::::::::::::::::::::::::::::::::
COMM MOVJ C00548 BC00548 VJ=30.00
COMM MOVL C00549 BC00549 V=666.7
COMM MOVL C00550 BC00550 V=250.0
COMM SFTON P0410
COMM MOVL C00551 BC00551 V=166.7 PL=0
COMM MACRO1 MJ#(0) ARGF24
COMM ARCON
COMM MOVL C00552 BC00552 V=7.5
COMM ARCOF
COMM MOVL C00553 BC00553 V=166.7
COMM SFTOF
COMM '------------------------
COMM 'W27.21
COMM '------------------------
COMM SFTON P0411
COMM MOVL C00554 BC00554 V=666.7
COMM MOVL C00555 BC00555 V=166.7 PL=0
COMM MACRO1 MJ#(0) ARGF24
COMM ARCON
COMM MOVL C00556 BC00556 V=7.5
COMM ARCOF
COMM MOVL C00557 BC00557 V=250.0
COMM SFTOF
COMM MOVJ C00558 BC00558 VJ=50.00
COMM MOVJ C00559 BC00559 VJ=50.00
COMM MOVJ C00560 BC00560 VJ=50.00
COMM '------------------------
COMM 'W27.22
COMM '------------------------
COMM MOVL C00561 BC00561 V=333.3
COMM MOVL C00562 BC00562 V=333.3
COMM SFTON P0412
COMM MOVL C00563 BC00563 V=166.7 PL=0
COMM MACRO1 MJ#(0) ARGF24
COMM ARCON
COMM MOVL C00564 BC00564 V=7.5
COMM ARCOF
COMM MOVL C00565 BC00565 V=200.0
COMM SFTOF
COMM '::::::::::::::::::::::::
COMM '::::::::::::::::::::::::
COMM '::::::::::::::::::::::::
COMM '::::::::::::::::::::::::
COMM '::::::::::::::::::::::::
COMM '::::::::::::::::::::::::
COMM '::::::::::::::::::::::::
COMM MOVJ C00566 BC00566 VJ=50.00
COMM MOVJ C00567 BC00567 VJ=50.00
COMM MOVJ C00568 BC00568 VJ=50.00
COMM MOVJ C00569 BC00569 VJ=50.00
MOVJ C00570 BC00570 VJ=50.00
'------------------------
'W215A
'------------------------
MOVJ C00571 BC00571 VJ=50.00
MOVJ C00572 BC00572 VJ=50.00
SFTON P0360
MOVL C00573 BC00573 V=500.0
MOVL C00574 BC00574 V=500.0
MOVL C00575 BC00575 V=166.7 PL=0
MACRO1 MJ#(0) ARGF9
ARCON
SFTOF
SFTON P0361
MOVL C00576 BC00576 V=11.7
MOVL C00577 BC00577 V=11.7
ARCOF
MOVL C00578 BC00578 V=500.0
SFTOF
MOVJ C00579 BC00579 VJ=50.00
MOVJ C00580 BC00580 VJ=50.00
MOVJ C00581 BC00581 VJ=50.00
MOVJ C00582 BC00582 VJ=80.00
MOVJ C00583 BC00583 VJ=50.00
MOVJ C00584 BC00584 VJ=50.00
MOVJ C00585 BC00585 VJ=40.00
MOVJ C00586 BC00586 VJ=20.00
MOVL C00587 BC00587 V=333.3
'------------------------
'W31.26
'------------------------
SFTON P0314
MOVL C00588 BC00588 V=833.3
MOVL C00589 BC00589 V=166.7 PL=0
MACRO1 MJ#(0) ARGF10
ARCON
MOVL C00590 BC00590 V=10.8
ARCOF
MOVL C00591 BC00591 V=200.0
SFTOF
'------------------------
'W31.27
'------------------------
SFTON P0315
MOVL C00592 BC00592 V=500.0
MOVL C00593 BC00593 V=166.7 PL=0
ARCON
MOVL C00594 BC00594 V=10.8
ARCOF
MOVL C00595 BC00595 V=200.0
SFTOF
MOVL C00596 BC00596 V=250.0
MOVL C00597 BC00597 V=250.0
MOVL C00598 BC00598 V=333.3
MOVL C00599 BC00599 V=416.7
MOVJ C00600 BC00600 VJ=30.00
MOVJ C00601 BC00601 VJ=30.00
MOVJ C00602 BC00602 VJ=50.00
MOVJ C00603 BC00603 VJ=50.00
COMM '::::::::::::::::::::::::
COMM '::::::::::::::::::::::::
COMM '::::::::::::::::::::::::
COMM '::::::::::::::::::::::::
COMM '::::::::::::::::::::::::
COMM '::::::::::::::::::::::::
COMM '::::::::::::::::::::::::
COMM MOVJ C00604 BC00604 VJ=50.00
COMM MOVJ C00605 BC00605 VJ=30.00
COMM MOVJ C00606 BC00606 VJ=30.00
COMM MOVJ C00607 BC00607 VJ=40.00
COMM MOVJ C00608 BC00608 VJ=50.00
COMM '::::::::::::::::::::::::::::::::
COMM '::::::::::::::::::::::::::::::::
COMM '------------------------
COMM 'W27.24
COMM '------------------------
COMM '::::::::::::::::::::::::::::::::
COMM '::::::::::::::::::::::::::::::::
COMM SFTON P0413
COMM MOVL C00609 BC00609 V=666.7
COMM MOVL C00610 BC00610 V=500.0
COMM MOVL C00611 BC00611 V=166.7 PL=0
COMM MACRO1 MJ#(0) ARGF24
COMM ARCON
COMM MOVL C00612 BC00612 V=7.5
COMM ARCOF
COMM MOVL C00613 BC00613 V=166.7
COMM SFTOF
COMM MOVJ C00614 BC00614 VJ=30.00
COMM MOVJ C00615 BC00615 VJ=30.00
COMM MOVJ C00616 BC00616 VJ=30.00
COMM '------------------------
COMM 'W27.26
COMM '------------------------
COMM SFTON P0414
COMM MOVL C00617 BC00617 V=333.3
COMM MOVL C00618 BC00618 V=333.3
COMM MOVL C00619 BC00619 V=166.7 PL=0
COMM MACRO1 MJ#(0) ARGF24
COMM ARCON
COMM MOVL C00620 BC00620 V=6.7
COMM ARCOF
COMM MOVL C00621 BC00621 V=200.0
SFTOF
COMM '------------------------
COMM 'W27.27
COMM '------------------------
COMM SFTON P0414
COMM MOVL C00622 BC00622 V=333.3
COMM MOVL C00623 BC00623 V=166.7 PL=0
COMM MACRO1 MJ#(0) ARGF24
COMM ARCON
COMM MOVL C00624 BC00624 V=6.7
COMM ARCOF
COMM MOVL C00625 BC00625 V=200.0
SFTOF
COMM MOVL C00626 BC00626 V=500.0
COMM '::::::::::::::::::::::::
COMM '::::::::::::::::::::::::
COMM '::::::::::::::::::::::::
COMM '::::::::::::::::::::::::
COMM '::::::::::::::::::::::::
COMM '::::::::::::::::::::::::
COMM '::::::::::::::::::::::::
COMM MOVL C00627 BC00627 V=833.3
COMM MOVJ C00628 BC00628 VJ=50.00
COMM MOVJ C00629 BC00629 VJ=50.00
COMM MOVJ C00630 BC00630 VJ=50.00
MOVJ C00631 BC00631 VJ=50.00
'------------------------
'W218A
'------------------------
MOVJ C00632 BC00632 VJ=50.00
MOVJ C00633 BC00633 VJ=50.00
SFTON P0357
MOVL C00634 BC00634 V=500.0
MOVL C00635 BC00635 V=500.0
MOVL C00636 BC00636 V=166.7 PL=0
MACRO1 MJ#(0) ARGF9
ARCON
SFTOF
SFTON P0356
MOVL C00637 BC00637 V=11.7
ARCOF
MOVL C00638 BC00638 V=333.3
SFTOF
MOVJ C00639 BC00639 VJ=50.00
MOVJ C00640 BC00640 VJ=50.00
MOVJ C00641 BC00641 VJ=50.00
MOVJ C00642 BC00642 VJ=50.00
MOVJ C00643 BC00643 VJ=50.00
MOVJ C00644 BC00644 VJ=50.00
MOVL C00645 BC00645 V=500.0
'------------------------
'W31.29
'------------------------
SFTON P0316
MOVL C00646 BC00646 V=333.3
MOVL C00647 BC00647 V=333.3
MOVL C00648 BC00648 V=166.7 PL=0
MOVL C00649 BC00649 V=166.7 PL=0
MACRO1 MJ#(0) ARGF10
ARCON
MOVL C00650 BC00650 V=10.8
ARCOF
MOVL C00651 BC00651 V=166.7
SFTOF
'------------------------
'W31.31
'------------------------
SFTON P0317
MOVL C00652 BC00652 V=666.7
MOVL C00653 BC00653 V=166.7 PL=0
MACRO1 MJ#(0) ARGF10
ARCON
MOVL C00654 BC00654 V=10.8
ARCOF
MOVL C00655 BC00655 V=166.7
SFTOF
'------------------------
'W31.32
'------------------------
SFTON P0317
MOVL C00656 BC00656 V=333.3
MOVL C00657 BC00657 V=166.7 PL=0
ARCON
MOVL C00658 BC00658 V=10.8
ARCOF
MOVL C00659 BC00659 V=166.7
SFTOF
MOVL C00660 BC00660 V=333.3
MOVL C00661 BC00661 V=416.7
MOVL C00662 BC00662 V=500.0
MOVL C00663 BC00663 V=500.0
MOVL C00664 BC00664 V=500.0
MOVJ C00665 BC00665 VJ=40.00
MOVJ C00666 BC00666 VJ=50.00
MOVJ C00667 BC00667 VJ=50.00
MOVJ C00668 BC00668 VJ=50.00
COMM '::::::::::::::::::::::::
COMM '::::::::::::::::::::::::
COMM '::::::::::::::::::::::::
COMM '::::::::::::::::::::::::
COMM '::::::::::::::::::::::::
COMM '::::::::::::::::::::::::
COMM '::::::::::::::::::::::::
COMM MOVJ C00669 BC00669 VJ=50.00
COMM MOVJ C00670 BC00670 VJ=50.00
COMM MOVJ C00671 BC00671 VJ=30.00
COMM '::::::::::::::::::::::::::::::::
COMM '::::::::::::::::::::::::::::::::
COMM '------------------------
COMM 'W27.29
COMM '------------------------
COMM '::::::::::::::::::::::::::::::::
COMM '::::::::::::::::::::::::::::::::
COMM SFTON P0416
COMM MOVL C00672 BC00672 V=666.7
COMM MOVL C00673 BC00673 V=166.7 PL=0
COMM MACRO1 MJ#(0) ARGF24
COMM ARCON
COMM MOVL C00674 BC00674 V=6.7
COMM ARCOF
COMM MOVL C00675 BC00675 V=166.7
COMM SFTOF
COMM '------------------------
COMM 'W27.31
COMM '------------------------
COMM SFTON P0417
COMM MOVL C00676 BC00676 V=666.7
COMM MOVL C00677 BC00677 V=166.7
COMM ARCON
COMM MOVL C00678 BC00678 V=7.5
COMM ARCOF
COMM MOVL C00679 BC00679 V=250.0
COMM SFTOF
COMM '------------------------
COMM 'W27.32
COMM '------------------------
COMM '::::::::::::::::::::::::
COMM '::::::::::::::::::::::::
COMM '::::::::::::::::::::::::
COMM '::::::::::::::::::::::::
COMM '::::::::::::::::::::::::
COMM '::::::::::::::::::::::::
COMM '::::::::::::::::::::::::
COMM MOVL C00680 BC00680 V=666.7
COMM MOVJ C00681 BC00681 VJ=40.00
COMM MOVJ C00682 BC00682 VJ=40.00
COMM MOVJ C00683 BC00683 VJ=40.00
COMM MOVJ C00684 BC00684 VJ=40.00
COMM MOVJ C00685 BC00685 VJ=50.00
COMM '------------------------
COMM 'W219A
COMM '------------------------
MOVJ C00686 BC00686 VJ=50.00
MOVJ C00687 BC00687 VJ=50.00
SFTON P0353
MOVL C00688 BC00688 V=666.7
MOVL C00689 BC00689 V=250.0
MOVL C00690 BC00690 V=166.7 PL=0
MACRO1 MJ#(0) ARGF9
ARCON
SFTOF
SFTON P0352
MOVL C00691 BC00691 V=11.7
ARCOF
MOVL C00692 BC00692 V=250.0
SFTOF
MOVJ C00693 BC00693 VJ=50.00
MOVJ C00694 BC00694 VJ=50.00
IFTHENEXP OT#(1457)=ON ANDEXP OT#(1441)=OFF
	 CALL JOB:TWIN_FRONT_WELD_-90ST-1_5340
ENDIF
IFTHENEXP OT#(1457)=OFF ANDEXP OT#(1441)=ON
	 CALL JOB:FRONT_WELD_-90ST-1_5340
ENDIF
CALL JOB:MOVE_OUT_OF_TUNNEL
END
